LIN {X 0,Y 656.609,Z 179.375,A -85,B 0,C 180,E1 30688.866,E2 30688.866} C_VEL
LIN {X 0,Y 656.676,Z 179.373,A -85,B 0,C 180,E1 30685.897,E2 30685.897} C_VEL
LIN {X 0,Y 656.608,Z 179.376,A -85,B 0,C 180,E1 30683.091,E2 30683.091} C_VEL
LIN {X 0,Y 656.674,Z 179.374,A -85,B 0,C 180,E1 30680.271,E2 30680.271} C_VEL
LIN {X 0,Y 656.609,Z 179.374,A -85,B 0,C 180,E1 30677.335,E2 30677.335} C_VEL
LIN {X 0,Y 656.626,Z 179.376,A -85,B 0,C 180,E1 30674.728,E2 30674.728} C_VEL
LIN {X 0,Y 656.62,Z 179.375,A -85,B 0,C 180,E1 30671.568,E2 30671.568} C_VEL
LIN {X 0,Y 656.615,Z 179.375,A -85,B 0,C 180,E1 30668.941,E2 30668.941} C_VEL
LIN {X 0,Y 656.649,Z 179.375,A -85,B 0,C 180,E1 30665.919,E2 30665.919} C_VEL
LIN {X 0,Y 656.609,Z 179.373,A -85,B 0,C 180,E1 30663.173,E2 30663.173} C_VEL
LIN {X 0,Y 656.682,Z 179.373,A -85,B 0,C 180,E1 30660.216,E2 30660.216} C_VEL
LIN {X 0,Y 656.607,Z 179.374,A -85,B 0,C 180,E1 30657.365,E2 30657.365} C_VEL
LIN {X 0,Y 656.689,Z 179.372,A -85,B 0,C 180,E1 30654.398,E2 30654.398} C_VEL
LIN {X 0,Y 656.607,Z 179.374,A -85,B 0,C 180,E1 30651.483,E2 30651.483} C_VEL
LIN {X 0,Y 656.656,Z 179.373,A -85,B 0,C 180,E1 30648.758,E2 30648.758} C_VEL
LIN {X 0,Y 656.615,Z 179.374,A -85,B 0,C 180,E1 30645.786,E2 30645.786} C_VEL
LIN {X 0,Y 656.622,Z 179.374,A -85,B 0,C 180,E1 30643.136,E2 30643.136} C_VEL
LIN {X 0,Y 656.625,Z 179.373,A -85,B 0,C 180,E1 30639.987,E2 30639.987} C_VEL
LIN {X 0,Y 656.612,Z 179.372,A -85,B 0,C 180,E1 30637.364,E2 30637.364} C_VEL
LIN {X 0,Y 656.649,Z 179.359,A -85,B 0,C 180,E1 30634.292,E2 30634.292} C_VEL
LIN {X 0,Y 656.61,Z 179.373,A -85,B 0,C 180,E1 30631.591,E2 30631.591} C_VEL
LIN {X 0,Y 656.691,Z 179.343,A -85,B 0,C 180,E1 30628.661,E2 30628.661} C_VEL
LIN {X 0,Y 656.607,Z 179.365,A -85,B 0,C 180,E1 30625.722,E2 30625.722} C_VEL
LIN {X 0,Y 656.697,Z 179.367,A -85,B 0,C 180,E1 30622.752,E2 30622.752} C_VEL
LIN {X 0,Y 656.608,Z 179.372,A -85,B 0,C 180,E1 30619.852,E2 30619.852} C_VEL
LIN {X 0,Y 656.666,Z 179.366,A -85,B 0,C 180,E1 30617.038,E2 30617.038} C_VEL
LIN {X 0,Y 656.612,Z 179.371,A -85,B 0,C 180,E1 30614.095,E2 30614.095} C_VEL
LIN {X 0,Y 656.628,Z 179.365,A -85,B 0,C 180,E1 30611.418,E2 30611.418} C_VEL
LIN {X 0,Y 656.622,Z 179.367,A -85,B 0,C 180,E1 30608.318,E2 30608.318} C_VEL
LIN {X 0,Y 656.609,Z 179.37,A -85,B 0,C 180,E1 30605.768,E2 30605.768} C_VEL
LIN {X 0,Y 656.67,Z 179.363,A -85,B 0,C 180,E1 30602.793,E2 30602.793} C_VEL
LIN {X 0,Y 656.607,Z 179.372,A -85,B 0,C 180,E1 30600,E2 30600} C_VEL
LIN {X 0,Y 656.686,Z 179.363,A -85,B 0,C 180,E1 30597.086,E2 30597.086} C_VEL
LIN {X 0,Y 656.609,Z 179.371,A -85,B 0,C 180,E1 30594.144,E2 30594.144} C_VEL
LIN {X 0,Y 656.641,Z 179.362,A -85,B 0,C 180,E1 30591.506,E2 30591.506} C_VEL
LIN {X 0,Y 656.614,Z 179.368,A -85,B 0,C 180,E1 30588.404,E2 30588.404} C_VEL
LIN {X 0,Y 656.628,Z 179.369,A -85,B 0,C 180,E1 30585.718,E2 30585.718} C_VEL
LIN {X 0,Y 656.62,Z 179.365,A -85,B 0,C 180,E1 30582.543,E2 30582.543} C_VEL
LIN {X 0,Y 656.621,Z 179.372,A -85,B 0,C 180,E1 30579.87,E2 30579.87} C_VEL
LIN {X 0,Y 656.624,Z 179.372,A -85,B 0,C 180,E1 30576.651,E2 30576.651} C_VEL
LIN {X 0,Y 656.618,Z 179.369,A -85,B 0,C 180,E1 30573.988,E2 30573.988} C_VEL
LIN {X 0,Y 656.631,Z 179.359,A -85,B 0,C 180,E1 30570.838,E2 30570.838} C_VEL
LIN {X 0,Y 656.612,Z 179.372,A -85,B 0,C 180,E1 30568.204,E2 30568.204} C_VEL
LIN {X 0,Y 656.678,Z 179.356,A -85,B 0,C 180,E1 30565.286,E2 30565.286} C_VEL
LIN {X 0,Y 656.609,Z 179.373,A -85,B 0,C 180,E1 30562.474,E2 30562.474} C_VEL
LIN {X 0,Y 656.666,Z 179.36,A -85,B 0,C 180,E1 30559.674,E2 30559.674} C_VEL
LIN {X 0,Y 656.612,Z 179.369,A -85,B 0,C 180,E1 30556.702,E2 30556.702} C_VEL
LIN {X 0,Y 656.639,Z 179.373,A -85,B 0,C 180,E1 30553.969,E2 30553.969} C_VEL
LIN {X 0,Y 656.622,Z 179.376,A -85,B 0,C 180,E1 30550.897,E2 30550.897} C_VEL
LIN {X 0,Y 656.614,Z 179.346,A -85,B 0,C 180,E1 30548.294,E2 30548.294} C_VEL
LIN {X 0,Y 656.638,Z 179.375,A -85,B 0,C 180,E1 30545.143,E2 30545.143} C_VEL
LIN {X 0,Y 656.711,Z 179.583,A -85,B 0,C 180,E1 30543.756,E2 30543.756} C_VEL
LIN {X 0,Y 663.323,Z 201.913,A -85,B 0,C 180,E1 30541.387,E2 30541.387} C_VEL
LIN {X 0,Y 662.57,Z 225.531,A -85,B 0,C 180,E1 30539.388,E2 30539.388} C_VEL
LIN {X 0,Y 667.017,Z 246.185,A -85,B 0,C 180,E1 30538.921,E2 30538.921} C_VEL
LIN {X 0,Y 664.801,Z 516.791,A -85,B 0,C 180,E1 30535.804,E2 30535.804} C_VEL
LIN {X 0,Y 664.373,Z 539.375,A -85,B 0,C 180,E1 30535.464,E2 30535.464} C_VEL
LIN {X 0,Y 663.94,Z 557.307,A -85,B 0,C 180,E1 30535.08,E2 30535.08} C_VEL
LIN {X 0,Y 663.439,Z 573.967,A -85,B 0,C 180,E1 30534.624,E2 30534.624} C_VEL
LIN {X 0,Y 662.861,Z 590.358,A -85,B 0,C 180,E1 30534.078,E2 30534.078} C_VEL
LIN {X 0,Y 662.199,Z 606.836,A -85,B 0,C 180,E1 30533.424,E2 30533.424} C_VEL
LIN {X 0,Y 661.522,Z 623.1,A -85,B 0,C 180,E1 30532.667,E2 30532.667} C_VEL
LIN {X 0,Y 660.779,Z 639.904,A -85,B 0,C 180,E1 30531.758,E2 30531.758} C_VEL
LIN {X 0,Y 659.792,Z 660.39,A -85,B 0,C 180,E1 30530.442,E2 30530.442} C_VEL
LIN {X 0,Y 659.062,Z 675.422,A -85,B 0,C 180,E1 30529.311,E2 30529.311} C_VEL
LIN {X 0,Y 658.429,Z 688.648,A -85,B 0,C 180,E1 30528.182,E2 30528.182} C_VEL
LIN {X 0,Y 657.872,Z 701.254,A -85,B 0,C 180,E1 30526.964,E2 30526.964} C_VEL
LIN {X 0,Y 657.324,Z 714.341,A -85,B 0,C 180,E1 30525.527,E2 30525.527} C_VEL
LIN {X 0,Y 656.796,Z 728.196,A -85,B 0,C 180,E1 30523.737,E2 30523.737} C_VEL
LIN {X 0,Y 656.462,Z 738.682,A -85,B 0,C 180,E1 30522.132,E2 30522.132} C_VEL
LIN {X 0,Y 656.245,Z 747.113,A -85,B 0,C 180,E1 30520.622,E2 30520.622} C_VEL
LIN {X 0,Y 656.073,Z 755.438,A -85,B 0,C 180,E1 30518.853,E2 30518.853} C_VEL
LIN {X 0,Y 655.962,Z 762.536,A -85,B 0,C 180,E1 30516.915,E2 30516.915} C_VEL
LIN {X 0,Y 655.927,Z 767.164,A -85,B 0,C 180,E1 30515.247,E2 30515.247} C_VEL
LIN {X 0,Y 655.919,Z 770.374,A -85,B 0,C 180,E1 30513.67,E2 30513.67} C_VEL
LIN {X 0,Y 655.916,Z 772.695,A -85,B 0,C 180,E1 30511.834,E2 30511.834} C_VEL
LIN {X 0,Y 655.903,Z 773.44,A -85,B 0,C 180,E1 30509.738,E2 30509.738} C_VEL
LIN {X 0,Y 655.913,Z 772.434,A -85,B 0,C 180,E1 30507.904,E2 30507.904} C_VEL
LIN {X 0,Y 655.922,Z 770.083,A -85,B 0,C 180,E1 30506.155,E2 30506.155} C_VEL
LIN {X 0,Y 655.941,Z 766.135,A -85,B 0,C 180,E1 30504.314,E2 30504.314} C_VEL
LIN {X 0,Y 655.999,Z 759.842,A -85,B 0,C 180,E1 30502.293,E2 30502.293} C_VEL
LIN {X 0,Y 656.109,Z 753.065,A -85,B 0,C 180,E1 30500.616,E2 30500.616} C_VEL
LIN {X 0,Y 656.274,Z 745.72,A -85,B 0,C 180,E1 30499.111,E2 30499.111} C_VEL
LIN {X 0,Y 656.555,Z 735.998,A -85,B 0,C 180,E1 30497.423,E2 30497.423} C_VEL
LIN {X 0,Y 656.97,Z 723.616,A -85,B 0,C 180,E1 30495.638,E2 30495.638} C_VEL
LIN {X 0,Y 657.408,Z 711.981,A -85,B 0,C 180,E1 30494.204,E2 30494.204} C_VEL
LIN {X 0,Y 657.918,Z 700.216,A -85,B 0,C 180,E1 30492.93,E2 30492.93} C_VEL
LIN {X 0,Y 658.499,Z 687.157,A -85,B 0,C 180,E1 30491.683,E2 30491.683} C_VEL
LIN {X 0,Y 659.331,Z 670.387,A -85,B 0,C 180,E1 30490.283,E2 30490.283} C_VEL
LIN {X 0,Y 660.165,Z 652.635,A -85,B 0,C 180,E1 30489.033,E2 30489.033} C_VEL
LIN {X 0,Y 660.876,Z 637.494,A -85,B 0,C 180,E1 30488.106,E2 30488.106} C_VEL
LIN {X 0,Y 661.557,Z 622.179,A -85,B 0,C 180,E1 30487.287,E2 30487.287} C_VEL
LIN {X 0,Y 662.229,Z 606.166,A -85,B 0,C 180,E1 30486.547,E2 30486.547} C_VEL
LIN {X 0,Y 662.861,Z 590.357,A -85,B 0,C 180,E1 30485.922,E2 30485.922} C_VEL
LIN {X 0,Y 663.439,Z 573.966,A -85,B 0,C 180,E1 30485.376,E2 30485.376} C_VEL
LIN {X 0,Y 663.961,Z 556.505,A -85,B 0,C 180,E1 30484.9,E2 30484.9} C_VEL
LIN {X 0,Y 664.453,Z 536.479,A -85,B 0,C 180,E1 30484.481,E2 30484.481} C_VEL
LIN {X 0,Y 664.876,Z 507.354,A -85,B 0,C 180,E1 30484.089,E2 30484.089} C_VEL
LIN {X 0,Y 667.019,Z 245.178,A -85,B 0,C 180,E1 30481.067,E2 30481.067} C_VEL
LIN {X 0,Y 662.536,Z 225.127,A -85,B 0,C 180,E1 30480.591,E2 30480.591} C_VEL
LIN {X 0,Y 663.211,Z 201.553,A -85,B 0,C 180,E1 30478.576,E2 30478.576} C_VEL
LIN {X 0,Y 656.698,Z 179.514,A -85,B 0,C 180,E1 30476.226,E2 30476.226} C_VEL
LIN {X 0,Y 656.607,Z 179.349,A -85,B 0,C 180,E1 30473.355,E2 30473.355} C_VEL
LIN {X 0,Y 656.694,Z 179.36,A -85,B 0,C 180,E1 30470.394,E2 30470.394} C_VEL
LIN {X 0,Y 656.609,Z 179.368,A -85,B 0,C 180,E1 30467.48,E2 30467.48} C_VEL
LIN {X 0,Y 656.686,Z 179.361,A -85,B 0,C 180,E1 30464.562,E2 30464.562} C_VEL
LIN {X 0,Y 656.611,Z 179.372,A -85,B 0,C 180,E1 30461.602,E2 30461.602} C_VEL
LIN {X 0,Y 656.657,Z 179.364,A -85,B 0,C 180,E1 30458.855,E2 30458.855} C_VEL
LIN {X 0,Y 656.617,Z 179.364,A -85,B 0,C 180,E1 30455.893,E2 30455.893} C_VEL
LIN {X 0,Y 656.622,Z 179.368,A -85,B 0,C 180,E1 30453.244,E2 30453.244} C_VEL
LIN {X 0,Y 656.625,Z 179.361,A -85,B 0,C 180,E1 30450.066,E2 30450.066} C_VEL
LIN {X 0,Y 656.614,Z 179.351,A -85,B 0,C 180,E1 30447.418,E2 30447.418} C_VEL
LIN {X 0,Y 656.65,Z 179.372,A -85,B 0,C 180,E1 30444.372,E2 30444.372} C_VEL
LIN {X 0,Y 656.607,Z 179.366,A -85,B 0,C 180,E1 30441.718,E2 30441.718} C_VEL
LIN {X 0,Y 656.689,Z 179.368,A -85,B 0,C 180,E1 30438.832,E2 30438.832} C_VEL
LIN {X 0,Y 656.609,Z 179.371,A -85,B 0,C 180,E1 30435.909,E2 30435.909} C_VEL
LIN {X 0,Y 656.636,Z 179.368,A -85,B 0,C 180,E1 30433.293,E2 30433.293} C_VEL
LIN {X 0,Y 656.616,Z 179.371,A -85,B 0,C 180,E1 30430.174,E2 30430.174} C_VEL
LIN {X 0,Y 656.621,Z 179.363,A -85,B 0,C 180,E1 30427.525,E2 30427.525} C_VEL
LIN {X 0,Y 656.625,Z 179.369,A -85,B 0,C 180,E1 30424.367,E2 30424.367} C_VEL
LIN {X 0,Y 656.612,Z 179.368,A -85,B 0,C 180,E1 30421.745,E2 30421.745} C_VEL
LIN {X 0,Y 656.664,Z 179.364,A -85,B 0,C 180,E1 30418.779,E2 30418.779} C_VEL
LIN {X 0,Y 656.606,Z 179.372,A -85,B 0,C 180,E1 30415.983,E2 30415.983} C_VEL
LIN {X 0,Y 656.691,Z 179.363,A -85,B 0,C 180,E1 30413.003,E2 30413.003} C_VEL
LIN {X 0,Y 656.608,Z 179.372,A -85,B 0,C 180,E1 30410.091,E2 30410.091} C_VEL
LIN {X 0,Y 656.69,Z 179.364,A -85,B 0,C 180,E1 30407.156,E2 30407.156} C_VEL
LIN {X 0,Y 656.608,Z 179.37,A -85,B 0,C 180,E1 30404.273,E2 30404.273} C_VEL
LIN {X 0,Y 656.65,Z 179.369,A -85,B 0,C 180,E1 30401.535,E2 30401.535} C_VEL
LIN {X 0,Y 656.614,Z 179.366,A -85,B 0,C 180,E1 30398.482,E2 30398.482} C_VEL
LIN {X 0,Y 656.619,Z 179.373,A -85,B 0,C 180,E1 30395.914,E2 30395.914} C_VEL
LIN {X 0,Y 656.622,Z 179.344,A -85,B 0,C 180,E1 30392.719,E2 30392.719} C_VEL
LIN {X 0,Y 656.61,Z 179.366,A -85,B 0,C 180,E1 30390.135,E2 30390.135} C_VEL
LIN {X 0,Y 656.67,Z 179.365,A -85,B 0,C 180,E1 30387.175,E2 30387.175} C_VEL
LIN {X 0,Y 656.603,Z 179.355,A -85,B 0,C 180,E1 30384.321,E2 30384.321} C_VEL
LIN {X 0,Y 656.691,Z 179.372,A -85,B 0,C 180,E1 30381.352,E2 30381.352} C_VEL
LIN {X 0,Y 656.608,Z 179.373,A -85,B 0,C 180,E1 30380.38,E2 30380.38} C_VEL
LIN {X 0,Y 655.64,Z 179.501,A -85,B 0,C 180,E1 30379.708,E2 30379.708} C_VEL
LIN {X 0,Y 649.202,Z 180.307,A -85,B 0,C 180,E1 30377.775,E2 30377.775} C_VEL
LIN {X 0,Y 648.739,Z 180.362,A -85,B 0,C 180,E1 30377.334,E2 30377.334} C_VEL
LIN {X 0,Y 648.669,Z 180.363,A -85,B 0,C 180,E1 30374.464,E2 30374.464} C_VEL
LIN {X 0,Y 648.756,Z 180.361,A -85,B 0,C 180,E1 30371.492,E2 30371.492} C_VEL
LIN {X 0,Y 648.668,Z 180.363,A -85,B 0,C 180,E1 30368.6,E2 30368.6} C_VEL
LIN {X 0,Y 648.743,Z 180.362,A -85,B 0,C 180,E1 30365.683,E2 30365.683} C_VEL
LIN {X 0,Y 648.669,Z 180.363,A -85,B 0,C 180,E1 30362.687,E2 30362.687} C_VEL
LIN {X 0,Y 648.741,Z 180.362,A -85,B 0,C 180,E1 30359.803,E2 30359.803} C_VEL
LIN {X 0,Y 648.67,Z 180.362,A -85,B 0,C 180,E1 30356.811,E2 30356.811} C_VEL
LIN {X 0,Y 648.721,Z 180.363,A -85,B 0,C 180,E1 30354.007,E2 30354.007} C_VEL
LIN {X 0,Y 648.676,Z 180.364,A -85,B 0,C 180,E1 30351.045,E2 30351.045} C_VEL
LIN {X 0,Y 648.691,Z 180.364,A -85,B 0,C 180,E1 30348.325,E2 30348.325} C_VEL
LIN {X 0,Y 648.68,Z 180.365,A -85,B 0,C 180,E1 30345.189,E2 30345.189} C_VEL
LIN {X 0,Y 648.677,Z 180.363,A -85,B 0,C 180,E1 30342.551,E2 30342.551} C_VEL
LIN {X 0,Y 648.692,Z 180.363,A -85,B 0,C 180,E1 30339.402,E2 30339.402} C_VEL
LIN {X 0,Y 648.671,Z 180.365,A -85,B 0,C 180,E1 30336.727,E2 30336.727} C_VEL
LIN {X 0,Y 648.72,Z 180.362,A -85,B 0,C 180,E1 30333.711,E2 30333.711} C_VEL
LIN {X 0,Y 648.669,Z 180.365,A -85,B 0,C 180,E1 30330.883,E2 30330.883} C_VEL
LIN {X 0,Y 648.747,Z 180.359,A -85,B 0,C 180,E1 30327.969,E2 30327.969} C_VEL
LIN {X 0,Y 648.668,Z 180.364,A -85,B 0,C 180,E1 30325.049,E2 30325.049} C_VEL
LIN {X 0,Y 648.756,Z 180.359,A -85,B 0,C 180,E1 30322.117,E2 30322.117} C_VEL
LIN {X 0,Y 648.669,Z 180.365,A -85,B 0,C 180,E1 30319.162,E2 30319.162} C_VEL
LIN {X 0,Y 648.755,Z 180.36,A -85,B 0,C 180,E1 30316.181,E2 30316.181} C_VEL
LIN {X 0,Y 648.669,Z 180.363,A -85,B 0,C 180,E1 30313.249,E2 30313.249} C_VEL
LIN {X 0,Y 648.742,Z 180.36,A -85,B 0,C 180,E1 30310.343,E2 30310.343} C_VEL
LIN {X 0,Y 648.672,Z 180.364,A -85,B 0,C 180,E1 30307.418,E2 30307.418} C_VEL
LIN {X 0,Y 648.699,Z 180.364,A -85,B 0,C 180,E1 30304.729,E2 30304.729} C_VEL
LIN {X 0,Y 648.679,Z 180.364,A -85,B 0,C 180,E1 30301.661,E2 30301.661} C_VEL
LIN {X 0,Y 648.673,Z 180.363,A -85,B 0,C 180,E1 30299.121,E2 30299.121} C_VEL
LIN {X 0,Y 648.718,Z 180.363,A -85,B 0,C 180,E1 30296.09,E2 30296.09} C_VEL
LIN {X 0,Y 648.672,Z 180.362,A -85,B 0,C 180,E1 30293.273,E2 30293.273} C_VEL
LIN {X 0,Y 648.735,Z 180.362,A -85,B 0,C 180,E1 30290.274,E2 30290.274} C_VEL
LIN {X 0,Y 648.669,Z 180.363,A -85,B 0,C 180,E1 30287.461,E2 30287.461} C_VEL
LIN {X 0,Y 648.748,Z 180.361,A -85,B 0,C 180,E1 30284.479,E2 30284.479} C_VEL
LIN {X 0,Y 648.671,Z 180.362,A -85,B 0,C 180,E1 30281.626,E2 30281.626} C_VEL
LIN {X 0,Y 648.713,Z 180.362,A -85,B 0,C 180,E1 30278.897,E2 30278.897} C_VEL
LIN {X 0,Y 648.671,Z 180.343,A -85,B 0,C 180,E1 30275.837,E2 30275.837} C_VEL
LIN {X 0,Y 648.688,Z 180.354,A -85,B 0,C 180,E1 30273.175,E2 30273.175} C_VEL
LIN {X 0,Y 648.683,Z 180.354,A -85,B 0,C 180,E1 30270.064,E2 30270.064} C_VEL
LIN {X 0,Y 648.674,Z 180.329,A -85,B 0,C 180,E1 30267.409,E2 30267.409} C_VEL
LIN {X 0,Y 648.701,Z 180.362,A -85,B 0,C 180,E1 30264.302,E2 30264.302} C_VEL
LIN {X 0,Y 648.669,Z 180.355,A -85,B 0,C 180,E1 30261.617,E2 30261.617} C_VEL
LIN {X 0,Y 648.744,Z 180.358,A -85,B 0,C 180,E1 30258.698,E2 30258.698} C_VEL
LIN {X 0,Y 648.667,Z 180.358,A -85,B 0,C 180,E1 30255.833,E2 30255.833} C_VEL
LIN {X 0,Y 648.738,Z 180.356,A -85,B 0,C 180,E1 30253.005,E2 30253.005} C_VEL
LIN {X 0,Y 648.671,Z 180.361,A -85,B 0,C 180,E1 30249.987,E2 30249.987} C_VEL
LIN {X 0,Y 648.723,Z 180.353,A -85,B 0,C 180,E1 30247.172,E2 30247.172} C_VEL
LIN {X 0,Y 648.671,Z 180.361,A -85,B 0,C 180,E1 30244.155,E2 30244.155} C_VEL
LIN {X 0,Y 648.7,Z 180.352,A -85,B 0,C 180,E1 30241.413,E2 30241.413} C_VEL
LIN {X 0,Y 648.677,Z 180.357,A -85,B 0,C 180,E1 30238.322,E2 30238.322} C_VEL
LIN {X 0,Y 648.69,Z 180.357,A -85,B 0,C 180,E1 30235.58,E2 30235.58} C_VEL
LIN {X 0,Y 648.682,Z 180.35,A -85,B 0,C 180,E1 30232.471,E2 30232.471} C_VEL
LIN {X 0,Y 648.679,Z 180.36,A -85,B 0,C 180,E1 30229.789,E2 30229.789} C_VEL
LIN {X 0,Y 648.691,Z 180.358,A -85,B 0,C 180,E1 30226.632,E2 30226.632} C_VEL
LIN {X 0,Y 648.672,Z 180.361,A -85,B 0,C 180,E1 30224.075,E2 30224.075} C_VEL
LIN {X 0,Y 648.743,Z 180.359,A -85,B 0,C 180,E1 30221.115,E2 30221.115} C_VEL
LIN {X 0,Y 648.67,Z 180.355,A -85,B 0,C 180,E1 30218.287,E2 30218.287} C_VEL
LIN {X 0,Y 648.742,Z 180.361,A -85,B 0,C 180,E1 30215.408,E2 30215.408} C_VEL
LIN {X 0,Y 648.669,Z 180.339,A -85,B 0,C 180,E1 30212.455,E2 30212.455} C_VEL
LIN {X 0,Y 648.705,Z 180.349,A -85,B 0,C 180,E1 30209.733,E2 30209.733} C_VEL
LIN {X 0,Y 648.678,Z 180.356,A -85,B 0,C 180,E1 30206.651,E2 30206.651} C_VEL
LIN {X 0,Y 648.691,Z 180.352,A -85,B 0,C 180,E1 30203.927,E2 30203.927} C_VEL
LIN {X 0,Y 648.681,Z 180.352,A -85,B 0,C 180,E1 30200.803,E2 30200.803} C_VEL
LIN {X 0,Y 648.676,Z 180.361,A -85,B 0,C 180,E1 30198.241,E2 30198.241} C_VEL
LIN {X 0,Y 648.71,Z 180.356,A -85,B 0,C 180,E1 30195.147,E2 30195.147} C_VEL
LIN {X 0,Y 648.672,Z 180.357,A -85,B 0,C 180,E1 30192.409,E2 30192.409} C_VEL
LIN {X 0,Y 648.742,Z 180.346,A -85,B 0,C 180,E1 30189.45,E2 30189.45} C_VEL
LIN {X 0,Y 648.668,Z 180.336,A -85,B 0,C 180,E1 30186.573,E2 30186.573} C_VEL
LIN {X 0,Y 648.721,Z 180.544,A -85,B 0,C 180,E1 30184.123,E2 30184.123} C_VEL
LIN {X 0,Y 655.582,Z 203.464,A -85,B 0,C 180,E1 30181.641,E2 30181.641} C_VEL
LIN {X 0,Y 655.853,Z 206.269,A -85,B 0,C 180,E1 30181.377,E2 30181.377} C_VEL
LIN {X 0,Y 655.176,Z 225.339,A -85,B 0,C 180,E1 30179.753,E2 30179.753} C_VEL
LIN {X 0,Y 659.991,Z 247.608,A -85,B 0,C 180,E1 30179.239,E2 30179.239} C_VEL
LIN {X 0,Y 657.572,Z 517.906,A -85,B 0,C 180,E1 30176.092,E2 30176.092} C_VEL
LIN {X 0,Y 657.117,Z 539.692,A -85,B 0,C 180,E1 30175.756,E2 30175.756} C_VEL
LIN {X 0,Y 656.647,Z 557.475,A -85,B 0,C 180,E1 30175.369,E2 30175.369} C_VEL
LIN {X 0,Y 656.088,Z 574.535,A -85,B 0,C 180,E1 30174.895,E2 30174.895} C_VEL
LIN {X 0,Y 655.488,Z 590.18,A -85,B 0,C 180,E1 30174.366,E2 30174.366} C_VEL
LIN {X 0,Y 654.779,Z 606.59,A -85,B 0,C 180,E1 30173.709,E2 30173.709} C_VEL
LIN {X 0,Y 654.071,Z 622.002,A -85,B 0,C 180,E1 30172.988,E2 30172.988} C_VEL
LIN {X 0,Y 653.293,Z 638.152,A -85,B 0,C 180,E1 30172.115,E2 30172.115} C_VEL
LIN {X 0,Y 652.35,Z 657.185,A -85,B 0,C 180,E1 30170.921,E2 30170.921} C_VEL
LIN {X 0,Y 651.442,Z 674.299,A -85,B 0,C 180,E1 30169.639,E2 30169.639} C_VEL
LIN {X 0,Y 650.738,Z 687.646,A -85,B 0,C 180,E1 30168.497,E2 30168.497} C_VEL
LIN {X 0,Y 650.113,Z 700.36,A -85,B 0,C 180,E1 30167.265,E2 30167.265} C_VEL
LIN {X 0,Y 649.567,Z 711.975,A -85,B 0,C 180,E1 30165.992,E2 30165.992} C_VEL
LIN {X 0,Y 649.058,Z 724.307,A -85,B 0,C 180,E1 30164.45,E2 30164.45} C_VEL
LIN {X 0,Y 648.597,Z 736.683,A -85,B 0,C 180,E1 30162.617,E2 30162.617} C_VEL
LIN {X 0,Y 648.311,Z 745.717,A -85,B 0,C 180,E1 30161.024,E2 30161.024} C_VEL
LIN {X 0,Y 648.131,Z 753.06,A -85,B 0,C 180,E1 30159.5,E2 30159.5} C_VEL
LIN {X 0,Y 648.01,Z 759.836,A -85,B 0,C 180,E1 30157.803,E2 30157.803} C_VEL
LIN {X 0,Y 647.947,Z 765.927,A -85,B 0,C 180,E1 30155.845,E2 30155.845} C_VEL
LIN {X 0,Y 647.923,Z 769.932,A -85,B 0,C 180,E1 30153.982,E2 30153.982} C_VEL
LIN {X 0,Y 647.909,Z 772.254,A -85,B 0,C 180,E1 30152.299,E2 30152.299} C_VEL
LIN {X 0,Y 647.903,Z 773.327,A -85,B 0,C 180,E1 30150.619,E2 30150.619} C_VEL
LIN {X 0,Y 647.902,Z 773.153,A -85,B 0,C 180,E1 30148.851,E2 30148.851} C_VEL
LIN {X 0,Y 647.904,Z 771.099,A -85,B 0,C 180,E1 30146.727,E2 30146.727} C_VEL
LIN {X 0,Y 647.917,Z 767.778,A -85,B 0,C 180,E1 30144.954,E2 30144.954} C_VEL
LIN {X 0,Y 647.958,Z 763.598,A -85,B 0,C 180,E1 30143.355,E2 30143.355} C_VEL
LIN {X 0,Y 648.049,Z 757.856,A -85,B 0,C 180,E1 30141.662,E2 30141.662} C_VEL
LIN {X 0,Y 648.235,Z 749.423,A -85,B 0,C 180,E1 30139.694,E2 30139.694} C_VEL
LIN {X 0,Y 648.489,Z 739.748,A -85,B 0,C 180,E1 30137.897,E2 30137.897} C_VEL
LIN {X 0,Y 648.822,Z 730.029,A -85,B 0,C 180,E1 30136.364,E2 30136.364} C_VEL
LIN {X 0,Y 649.247,Z 719.431,A -85,B 0,C 180,E1 30134.916,E2 30134.916} C_VEL
LIN {X 0,Y 649.876,Z 705.645,A -85,B 0,C 180,E1 30133.281,E2 30133.281} C_VEL
LIN {X 0,Y 650.594,Z 690.538,A -85,B 0,C 180,E1 30131.769,E2 30131.769} C_VEL
LIN {X 0,Y 651.287,Z 677.089,A -85,B 0,C 180,E1 30130.589,E2 30130.589} C_VEL
LIN {X 0,Y 651.98,Z 663.838,A -85,B 0,C 180,E1 30129.561,E2 30129.561} C_VEL
LIN {X 0,Y 652.719,Z 649.399,A -85,B 0,C 180,E1 30128.574,E2 30128.574} C_VEL
LIN {X 0,Y 653.476,Z 634.276,A -85,B 0,C 180,E1 30127.664,E2 30127.664} C_VEL
LIN {X 0,Y 654.308,Z 617.395,A -85,B 0,C 180,E1 30126.783,E2 30126.783} C_VEL
LIN {X 0,Y 655.285,Z 595.284,A -85,B 0,C 180,E1 30125.822,E2 30125.822} C_VEL
LIN {X 0,Y 656.006,Z 576.766,A -85,B 0,C 180,E1 30125.174,E2 30125.174} C_VEL
LIN {X 0,Y 656.593,Z 559.359,A -85,B 0,C 180,E1 30124.679,E2 30124.679} C_VEL
LIN {X 0,Y 657.058,Z 542.385,A -85,B 0,C 180,E1 30124.297,E2 30124.297} C_VEL
LIN {X 0,Y 657.429,Z 525.016,A -85,B 0,C 180,E1 30124.007,E2 30124.007} C_VEL
LIN {X 0,Y 659.812,Z 267.465,A -85,B 0,C 180,E1 30120.995,E2 30120.995} C_VEL
LIN {X 0,Y 659.802,Z 245.831,A -85,B 0,C 180,E1 30120.73,E2 30120.73} C_VEL
LIN {X 0,Y 655.119,Z 224.707,A -85,B 0,C 180,E1 30120.216,E2 30120.216} C_VEL
LIN {X 0,Y 655.742,Z 204.05,A -85,B 0,C 180,E1 30118.419,E2 30118.419} C_VEL
LIN {X 0,Y 649.083,Z 181.929,A -85,B 0,C 180,E1 30116.052,E2 30116.052} C_VEL
LIN {X 0,Y 648.713,Z 180.503,A -85,B 0,C 180,E1 30115.864,E2 30115.864} C_VEL
LIN {X 0,Y 648.674,Z 180.329,A -85,B 0,C 180,E1 30113.131,E2 30113.131} C_VEL
LIN {X 0,Y 648.702,Z 180.366,A -85,B 0,C 180,E1 30110.002,E2 30110.002} C_VEL
LIN {X 0,Y 648.673,Z 180.357,A -85,B 0,C 180,E1 30107.302,E2 30107.302} C_VEL
LIN {X 0,Y 648.73,Z 180.35,A -85,B 0,C 180,E1 30104.284,E2 30104.284} C_VEL
LIN {X 0,Y 648.671,Z 180.361,A -85,B 0,C 180,E1 30101.493,E2 30101.493} C_VEL
LIN {X 0,Y 648.756,Z 180.352,A -85,B 0,C 180,E1 30098.62,E2 30098.62} C_VEL
LIN {X 0,Y 648.669,Z 180.352,A -85,B 0,C 180,E1 30095.639,E2 30095.639} C_VEL
LIN {X 0,Y 648.748,Z 180.357,A -85,B 0,C 180,E1 30092.71,E2 30092.71} C_VEL
LIN {X 0,Y 648.67,Z 180.349,A -85,B 0,C 180,E1 30089.759,E2 30089.759} C_VEL
LIN {X 0,Y 648.722,Z 180.339,A -85,B 0,C 180,E1 30086.946,E2 30086.946} C_VEL
LIN {X 0,Y 648.674,Z 180.361,A -85,B 0,C 180,E1 30083.916,E2 30083.916} C_VEL
LIN {X 0,Y 648.695,Z 180.354,A -85,B 0,C 180,E1 30081.237,E2 30081.237} C_VEL
LIN {X 0,Y 648.683,Z 180.353,A -85,B 0,C 180,E1 30078.142,E2 30078.142} C_VEL
LIN {X 0,Y 648.682,Z 180.359,A -85,B 0,C 180,E1 30075.466,E2 30075.466} C_VEL
LIN {X 0,Y 648.686,Z 180.357,A -85,B 0,C 180,E1 30072.28,E2 30072.28} C_VEL
LIN {X 0,Y 648.678,Z 180.36,A -85,B 0,C 180,E1 30069.583,E2 30069.583} C_VEL
LIN {X 0,Y 648.697,Z 180.361,A -85,B 0,C 180,E1 30066.461,E2 30066.461} C_VEL
LIN {X 0,Y 648.67,Z 180.358,A -85,B 0,C 180,E1 30063.801,E2 30063.801} C_VEL
LIN {X 0,Y 648.731,Z 180.361,A -85,B 0,C 180,E1 30060.795,E2 30060.795} C_VEL
LIN {X 0,Y 648.668,Z 180.353,A -85,B 0,C 180,E1 30057.968,E2 30057.968} C_VEL
LIN {X 0,Y 648.749,Z 180.361,A -85,B 0,C 180,E1 30055.049,E2 30055.049} C_VEL
LIN {X 0,Y 648.67,Z 180.356,A -85,B 0,C 180,E1 30052.204,E2 30052.204} C_VEL
LIN {X 0,Y 648.715,Z 180.361,A -85,B 0,C 180,E1 30049.431,E2 30049.431} C_VEL
LIN {X 0,Y 648.673,Z 180.361,A -85,B 0,C 180,E1 30046.359,E2 30046.359} C_VEL
LIN {X 0,Y 648.683,Z 180.359,A -85,B 0,C 180,E1 30043.775,E2 30043.775} C_VEL
LIN {X 0,Y 648.68,Z 180.361,A -85,B 0,C 180,E1 30040.552,E2 30040.552} C_VEL
LIN {X 0,Y 648.683,Z 180.355,A -85,B 0,C 180,E1 30037.86,E2 30037.86} C_VEL
LIN {X 0,Y 648.681,Z 180.354,A -85,B 0,C 180,E1 30034.627,E2 30034.627} C_VEL
LIN {X 0,Y 648.679,Z 180.331,A -85,B 0,C 180,E1 30031.957,E2 30031.957} C_VEL
LIN {X 0,Y 648.689,Z 180.362,A -85,B 0,C 180,E1 30028.8,E2 30028.8} C_VEL
LIN {X 0,Y 648.673,Z 180.353,A -85,B 0,C 180,E1 30026.173,E2 30026.173} C_VEL
LIN {X 0,Y 648.716,Z 180.356,A -85,B 0,C 180,E1 30023.115,E2 30023.115} C_VEL
LIN {X 0,Y 648.67,Z 180.362,A -85,B 0,C 180,E1 30020.345,E2 30020.345} C_VEL
LIN {X 0,Y 648.748,Z 180.361,A -85,B 0,C 180,E1 30017.42,E2 30017.42} C_VEL
LIN {X 0,Y 648.739,Z 180.362,A -85,B 0,C 180,E1 30017.334,E2 30017.334} C_VEL
LIN {X 0,Y 647.695,Z 180.49,A -85,B 0,C 180,E1 30016.653,E2 30016.653} C_VEL
LIN {X 0,Y 641.24,Z 181.29,A -85,B 0,C 180,E1 30014.746,E2 30014.746} C_VEL
LIN {X 0,Y 640.736,Z 181.352,A -85,B 0,C 180,E1 30014.25,E2 30014.25} C_VEL
LIN {X 0,Y 640.769,Z 181.351,A -85,B 0,C 180,E1 30011.179,E2 30011.179} C_VEL
LIN {X 0,Y 640.732,Z 181.352,A -85,B 0,C 180,E1 30008.427,E2 30008.427} C_VEL
LIN {X 0,Y 640.798,Z 181.35,A -85,B 0,C 180,E1 30005.46,E2 30005.46} C_VEL
LIN {X 0,Y 640.731,Z 181.353,A -85,B 0,C 180,E1 30002.569,E2 30002.569} C_VEL
LIN {X 0,Y 640.818,Z 181.347,A -85,B 0,C 180,E1 29999.641,E2 29999.641} C_VEL
LIN {X 0,Y 640.731,Z 181.352,A -85,B 0,C 180,E1 29996.704,E2 29996.704} C_VEL
LIN {X 0,Y 640.813,Z 181.348,A -85,B 0,C 180,E1 29993.735,E2 29993.735} C_VEL
LIN {X 0,Y 640.73,Z 181.353,A -85,B 0,C 180,E1 29990.809,E2 29990.809} C_VEL
LIN {X 0,Y 640.808,Z 181.349,A -85,B 0,C 180,E1 29987.857,E2 29987.857} C_VEL
LIN {X 0,Y 640.73,Z 181.354,A -85,B 0,C 180,E1 29984.919,E2 29984.919} C_VEL
LIN {X 0,Y 640.789,Z 181.352,A -85,B 0,C 180,E1 29982.068,E2 29982.068} C_VEL
LIN {X 0,Y 640.732,Z 181.353,A -85,B 0,C 180,E1 29979.067,E2 29979.067} C_VEL
LIN {X 0,Y 640.76,Z 181.354,A -85,B 0,C 180,E1 29976.36,E2 29976.36} C_VEL
LIN {X 0,Y 640.736,Z 181.354,A -85,B 0,C 180,E1 29973.22,E2 29973.22} C_VEL
LIN {X 0,Y 640.757,Z 181.352,A -85,B 0,C 180,E1 29970.447,E2 29970.447} C_VEL
LIN {X 0,Y 640.737,Z 181.354,A -85,B 0,C 180,E1 29967.317,E2 29967.317} C_VEL
LIN {X 0,Y 640.757,Z 181.353,A -85,B 0,C 180,E1 29964.539,E2 29964.539} C_VEL
LIN {X 0,Y 640.737,Z 181.353,A -85,B 0,C 180,E1 29961.385,E2 29961.385} C_VEL
LIN {X 0,Y 640.751,Z 181.354,A -85,B 0,C 180,E1 29958.662,E2 29958.662} C_VEL
LIN {X 0,Y 640.744,Z 181.354,A -85,B 0,C 180,E1 29955.543,E2 29955.543} C_VEL
LIN {X 0,Y 640.741,Z 181.353,A -85,B 0,C 180,E1 29952.849,E2 29952.849} C_VEL
LIN {X 0,Y 640.746,Z 181.353,A -85,B 0,C 180,E1 29949.638,E2 29949.638} C_VEL
LIN {X 0,Y 640.737,Z 181.353,A -85,B 0,C 180,E1 29947.031,E2 29947.031} C_VEL
LIN {X 0,Y 640.778,Z 181.351,A -85,B 0,C 180,E1 29943.997,E2 29943.997} C_VEL
LIN {X 0,Y 640.733,Z 181.353,A -85,B 0,C 180,E1 29941.175,E2 29941.175} C_VEL
LIN {X 0,Y 640.793,Z 181.35,A -85,B 0,C 180,E1 29938.174,E2 29938.174} C_VEL
LIN {X 0,Y 640.73,Z 181.353,A -85,B 0,C 180,E1 29935.327,E2 29935.327} C_VEL
LIN {X 0,Y 640.801,Z 181.35,A -85,B 0,C 180,E1 29932.296,E2 29932.296} C_VEL
LIN {X 0,Y 640.731,Z 181.351,A -85,B 0,C 180,E1 29929.463,E2 29929.463} C_VEL
LIN {X 0,Y 640.809,Z 181.349,A -85,B 0,C 180,E1 29926.516,E2 29926.516} C_VEL
LIN {X 0,Y 640.732,Z 181.352,A -85,B 0,C 180,E1 29923.611,E2 29923.611} C_VEL
LIN {X 0,Y 640.801,Z 181.351,A -85,B 0,C 180,E1 29920.691,E2 29920.691} C_VEL
LIN {X 0,Y 640.732,Z 181.35,A -85,B 0,C 180,E1 29917.713,E2 29917.713} C_VEL
LIN {X 0,Y 640.784,Z 181.324,A -85,B 0,C 180,E1 29914.828,E2 29914.828} C_VEL
LIN {X 0,Y 640.733,Z 181.351,A -85,B 0,C 180,E1 29911.834,E2 29911.834} C_VEL
LIN {X 0,Y 640.758,Z 181.337,A -85,B 0,C 180,E1 29909.135,E2 29909.135} C_VEL
LIN {X 0,Y 640.739,Z 181.342,A -85,B 0,C 180,E1 29906.007,E2 29906.007} C_VEL
LIN {X 0,Y 640.757,Z 181.351,A -85,B 0,C 180,E1 29903.22,E2 29903.22} C_VEL
LIN {X 0,Y 640.739,Z 181.35,A -85,B 0,C 180,E1 29900.064,E2 29900.064} C_VEL
LIN {X 0,Y 640.752,Z 181.346,A -85,B 0,C 180,E1 29897.341,E2 29897.341} C_VEL
LIN {X 0,Y 640.74,Z 181.349,A -85,B 0,C 180,E1 29894.182,E2 29894.182} C_VEL
LIN {X 0,Y 640.75,Z 181.342,A -85,B 0,C 180,E1 29891.431,E2 29891.431} C_VEL
LIN {X 0,Y 640.74,Z 181.344,A -85,B 0,C 180,E1 29888.254,E2 29888.254} C_VEL
LIN {X 0,Y 640.737,Z 181.348,A -85,B 0,C 180,E1 29885.642,E2 29885.642} C_VEL
LIN {X 0,Y 640.756,Z 181.34,A -85,B 0,C 180,E1 29882.504,E2 29882.504} C_VEL
LIN {X 0,Y 640.733,Z 181.35,A -85,B 0,C 180,E1 29879.821,E2 29879.821} C_VEL
LIN {X 0,Y 640.782,Z 181.343,A -85,B 0,C 180,E1 29876.78,E2 29876.78} C_VEL
LIN {X 0,Y 640.731,Z 181.349,A -85,B 0,C 180,E1 29873.998,E2 29873.998} C_VEL
LIN {X 0,Y 640.807,Z 181.343,A -85,B 0,C 180,E1 29871.023,E2 29871.023} C_VEL
LIN {X 0,Y 640.73,Z 181.346,A -85,B 0,C 180,E1 29868.112,E2 29868.112} C_VEL
LIN {X 0,Y 640.823,Z 181.347,A -85,B 0,C 180,E1 29865.173,E2 29865.173} C_VEL
LIN {X 0,Y 640.731,Z 181.342,A -85,B 0,C 180,E1 29862.19,E2 29862.19} C_VEL
LIN {X 0,Y 640.814,Z 181.346,A -85,B 0,C 180,E1 29859.256,E2 29859.256} C_VEL
LIN {X 0,Y 640.732,Z 181.35,A -85,B 0,C 180,E1 29856.336,E2 29856.336} C_VEL
LIN {X 0,Y 640.807,Z 181.33,A -85,B 0,C 180,E1 29853.376,E2 29853.376} C_VEL
LIN {X 0,Y 640.732,Z 181.338,A -85,B 0,C 180,E1 29850.453,E2 29850.453} C_VEL
LIN {X 0,Y 640.77,Z 181.351,A -85,B 0,C 180,E1 29847.741,E2 29847.741} C_VEL
LIN {X 0,Y 640.738,Z 181.34,A -85,B 0,C 180,E1 29844.691,E2 29844.691} C_VEL
LIN {X 0,Y 640.754,Z 181.352,A -85,B 0,C 180,E1 29841.946,E2 29841.946} C_VEL
LIN {X 0,Y 640.741,Z 181.35,A -85,B 0,C 180,E1 29838.77,E2 29838.77} C_VEL
LIN {X 0,Y 640.757,Z 181.343,A -85,B 0,C 180,E1 29835.995,E2 29835.995} C_VEL
LIN {X 0,Y 640.739,Z 181.346,A -85,B 0,C 180,E1 29832.823,E2 29832.823} C_VEL
LIN {X 0,Y 640.751,Z 181.355,A -85,B 0,C 180,E1 29830.12,E2 29830.12} C_VEL
LIN {X 0,Y 640.738,Z 181.314,A -85,B 0,C 180,E1 29826.922,E2 29826.922} C_VEL
LIN {X 0,Y 640.756,Z 181.506,A -85,B 0,C 180,E1 29824.498,E2 29824.498} C_VEL
LIN {X 0,Y 646.698,Z 200.886,A -85,B 0,C 180,E1 29822.337,E2 29822.337} C_VEL
LIN {X 0,Y 648.463,Z 207.835,A -85,B 0,C 180,E1 29821.614,E2 29821.614} C_VEL
LIN {X 0,Y 647.799,Z 225.092,A -85,B 0,C 180,E1 29820.128,E2 29820.128} C_VEL
LIN {X 0,Y 652.986,Z 249.076,A -85,B 0,C 180,E1 29819.563,E2 29819.563} C_VEL
LIN {X 0,Y 650.351,Z 519.06,A -85,B 0,C 180,E1 29816.384,E2 29816.384} C_VEL
LIN {X 0,Y 649.882,Z 539.793,A -85,B 0,C 180,E1 29816.058,E2 29816.058} C_VEL
LIN {X 0,Y 649.377,Z 557.413,A -85,B 0,C 180,E1 29815.67,E2 29815.67} C_VEL
LIN {X 0,Y 648.786,Z 574.205,A -85,B 0,C 180,E1 29815.199,E2 29815.199} C_VEL
LIN {X 0,Y 648.119,Z 590.337,A -85,B 0,C 180,E1 29814.649,E2 29814.649} C_VEL
LIN {X 0,Y 647.389,Z 606.088,A -85,B 0,C 180,E1 29814.011,E2 29814.011} C_VEL
LIN {X 0,Y 646.602,Z 621.823,A -85,B 0,C 180,E1 29813.269,E2 29813.269} C_VEL
LIN {X 0,Y 645.755,Z 637.974,A -85,B 0,C 180,E1 29812.387,E2 29812.387} C_VEL
LIN {X 0,Y 644.738,Z 657.006,A -85,B 0,C 180,E1 29811.18,E2 29811.18} C_VEL
LIN {X 0,Y 643.754,Z 674.156,A -85,B 0,C 180,E1 29809.883,E2 29809.883} C_VEL
LIN {X 0,Y 643.011,Z 687.486,A -85,B 0,C 180,E1 29808.736,E2 29808.736} C_VEL
LIN {X 0,Y 642.365,Z 699.466,A -85,B 0,C 180,E1 29807.574,E2 29807.574} C_VEL
LIN {X 0,Y 641.771,Z 711.183,A -85,B 0,C 180,E1 29806.284,E2 29806.284} C_VEL
LIN {X 0,Y 641.252,Z 722.212,A -85,B 0,C 180,E1 29804.907,E2 29804.907} C_VEL
LIN {X 0,Y 640.78,Z 733.705,A -85,B 0,C 180,E1 29803.259,E2 29803.259} C_VEL
LIN {X 0,Y 640.383,Z 744.785,A -85,B 0,C 180,E1 29801.345,E2 29801.345} C_VEL
LIN {X 0,Y 640.173,Z 752.503,A -85,B 0,C 180,E1 29799.746,E2 29799.746} C_VEL
LIN {X 0,Y 640.051,Z 758.839,A -85,B 0,C 180,E1 29798.172,E2 29798.172} C_VEL
LIN {X 0,Y 639.961,Z 764.126,A -85,B 0,C 180,E1 29796.548,E2 29796.548} C_VEL
LIN {X 0,Y 639.92,Z 768.802,A -85,B 0,C 180,E1 29794.66,E2 29794.66} C_VEL
LIN {X 0,Y 639.911,Z 771.986,A -85,B 0,C 180,E1 29792.597,E2 29792.597} C_VEL
LIN {X 0,Y 639.91,Z 773.265,A -85,B 0,C 180,E1 29790.806,E2 29790.806} C_VEL
LIN {X 0,Y 639.91,Z 773.265,A -85,B 0,C 180,E1 29789.194,E2 29789.194} C_VEL
LIN {X 0,Y 639.911,Z 771.986,A -85,B 0,C 180,E1 29787.403,E2 29787.403} C_VEL
LIN {X 0,Y 639.92,Z 768.802,A -85,B 0,C 180,E1 29785.34,E2 29785.34} C_VEL
LIN {X 0,Y 639.961,Z 764.126,A -85,B 0,C 180,E1 29783.452,E2 29783.452} C_VEL
LIN {X 0,Y 640.051,Z 758.839,A -85,B 0,C 180,E1 29781.828,E2 29781.828} C_VEL
LIN {X 0,Y 640.173,Z 752.503,A -85,B 0,C 180,E1 29780.254,E2 29780.254} C_VEL
LIN {X 0,Y 640.383,Z 744.785,A -85,B 0,C 180,E1 29778.655,E2 29778.655} C_VEL
LIN {X 0,Y 640.78,Z 733.705,A -85,B 0,C 180,E1 29776.741,E2 29776.741} C_VEL
LIN {X 0,Y 641.252,Z 722.212,A -85,B 0,C 180,E1 29775.093,E2 29775.093} C_VEL
LIN {X 0,Y 641.77,Z 711.182,A -85,B 0,C 180,E1 29773.716,E2 29773.716} C_VEL
LIN {X 0,Y 642.365,Z 699.465,A -85,B 0,C 180,E1 29772.426,E2 29772.426} C_VEL
LIN {X 0,Y 643.036,Z 687.079,A -85,B 0,C 180,E1 29771.226,E2 29771.226} C_VEL
LIN {X 0,Y 643.918,Z 671.351,A -85,B 0,C 180,E1 29769.885,E2 29769.885} C_VEL
LIN {X 0,Y 644.95,Z 652.778,A -85,B 0,C 180,E1 29768.541,E2 29768.541} C_VEL
LIN {X 0,Y 645.789,Z 637.242,A -85,B 0,C 180,E1 29767.571,E2 29767.571} C_VEL
LIN {X 0,Y 646.623,Z 621.425,A -85,B 0,C 180,E1 29766.711,E2 29766.711} C_VEL
LIN {X 0,Y 647.389,Z 606.088,A -85,B 0,C 180,E1 29765.989,E2 29765.989} C_VEL
LIN {X 0,Y 648.158,Z 589.426,A -85,B 0,C 180,E1 29765.317,E2 29765.317} C_VEL
LIN {X 0,Y 648.867,Z 572.128,A -85,B 0,C 180,E1 29764.736,E2 29764.736} C_VEL
LIN {X 0,Y 649.617,Z 550.932,A -85,B 0,C 180,E1 29764.167,E2 29764.167} C_VEL
LIN {X 0,Y 650.177,Z 528.3,A -85,B 0,C 180,E1 29763.747,E2 29763.747} C_VEL
LIN {X 0,Y 650.738,Z 478.737,A -85,B 0,C 180,E1 29763.141,E2 29763.141} C_VEL
LIN {X 0,Y 652.877,Z 247.678,A -85,B 0,C 180,E1 29760.414,E2 29760.414} C_VEL
LIN {X 0,Y 647.738,Z 224.416,A -85,B 0,C 180,E1 29759.839,E2 29759.839} C_VEL
LIN {X 0,Y 648.331,Z 206.708,A -85,B 0,C 180,E1 29758.275,E2 29758.275} C_VEL
LIN {X 0,Y 641.323,Z 183.497,A -85,B 0,C 180,E1 29755.753,E2 29755.753} C_VEL
LIN {X 0,Y 640.749,Z 181.471,A -85,B 0,C 180,E1 29755.482,E2 29755.482} C_VEL
LIN {X 0,Y 640.789,Z 181.303,A -85,B 0,C 180,E1 29752.585,E2 29752.585} C_VEL
LIN {X 0,Y 640.735,Z 181.355,A -85,B 0,C 180,E1 29749.601,E2 29749.601} C_VEL
LIN {X 0,Y 640.763,Z 181.345,A -85,B 0,C 180,E1 29746.891,E2 29746.891} C_VEL
LIN {X 0,Y 640.744,Z 181.346,A -85,B 0,C 180,E1 29743.858,E2 29743.858} C_VEL
LIN {X 0,Y 640.752,Z 181.35,A -85,B 0,C 180,E1 29741.095,E2 29741.095} C_VEL
LIN {X 0,Y 640.745,Z 181.352,A -85,B 0,C 180,E1 29737.941,E2 29737.941} C_VEL
LIN {X 0,Y 640.741,Z 181.34,A -85,B 0,C 180,E1 29735.268,E2 29735.268} C_VEL
LIN {X 0,Y 640.749,Z 181.35,A -85,B 0,C 180,E1 29732.044,E2 29732.044} C_VEL
LIN {X 0,Y 640.735,Z 181.338,A -85,B 0,C 180,E1 29729.444,E2 29729.444} C_VEL
LIN {X 0,Y 640.778,Z 181.34,A -85,B 0,C 180,E1 29726.406,E2 29726.406} C_VEL
LIN {X 0,Y 640.733,Z 181.35,A -85,B 0,C 180,E1 29723.645,E2 29723.645} C_VEL
LIN {X 0,Y 640.805,Z 181.348,A -85,B 0,C 180,E1 29720.649,E2 29720.649} C_VEL
LIN {X 0,Y 640.733,Z 181.341,A -85,B 0,C 180,E1 29717.717,E2 29717.717} C_VEL
LIN {X 0,Y 640.801,Z 181.345,A -85,B 0,C 180,E1 29714.693,E2 29714.693} C_VEL
LIN {X 0,Y 640.731,Z 181.346,A -85,B 0,C 180,E1 29711.796,E2 29711.796} C_VEL
LIN {X 0,Y 640.805,Z 181.339,A -85,B 0,C 180,E1 29708.796,E2 29708.796} C_VEL
LIN {X 0,Y 640.731,Z 181.35,A -85,B 0,C 180,E1 29705.912,E2 29705.912} C_VEL
LIN {X 0,Y 640.809,Z 181.339,A -85,B 0,C 180,E1 29702.952,E2 29702.952} C_VEL
LIN {X 0,Y 640.73,Z 181.35,A -85,B 0,C 180,E1 29700,E2 29700} C_VEL
LIN {X 0,Y 640.808,Z 181.34,A -85,B 0,C 180,E1 29697.048,E2 29697.048} C_VEL
LIN {X 0,Y 640.73,Z 181.348,A -85,B 0,C 180,E1 29694.088,E2 29694.088} C_VEL
LIN {X 0,Y 640.804,Z 181.345,A -85,B 0,C 180,E1 29691.204,E2 29691.204} C_VEL
LIN {X 0,Y 640.73,Z 181.343,A -85,B 0,C 180,E1 29688.204,E2 29688.204} C_VEL
LIN {X 0,Y 640.804,Z 181.35,A -85,B 0,C 180,E1 29685.265,E2 29685.265} C_VEL
LIN {X 0,Y 640.732,Z 181.346,A -85,B 0,C 180,E1 29682.284,E2 29682.284} C_VEL
LIN {X 0,Y 640.802,Z 181.346,A -85,B 0,C 180,E1 29679.351,E2 29679.351} C_VEL
LIN {X 0,Y 640.731,Z 181.351,A -85,B 0,C 180,E1 29676.355,E2 29676.355} C_VEL
LIN {X 0,Y 640.788,Z 181.328,A -85,B 0,C 180,E1 29673.495,E2 29673.495} C_VEL
LIN {X 0,Y 640.734,Z 181.343,A -85,B 0,C 180,E1 29670.536,E2 29670.536} C_VEL
LIN {X 0,Y 640.749,Z 181.351,A -85,B 0,C 180,E1 29667.912,E2 29667.912} C_VEL
LIN {X 0,Y 640.737,Z 181.328,A -85,B 0,C 180,E1 29664.732,E2 29664.732} C_VEL
LIN {X 0,Y 640.748,Z 181.35,A -85,B 0,C 180,E1 29661.994,E2 29661.994} C_VEL
LIN {X 0,Y 640.741,Z 181.351,A -85,B 0,C 180,E1 29658.77,E2 29658.77} C_VEL
LIN {X 0,Y 640.755,Z 181.352,A -85,B 0,C 180,E1 29655.996,E2 29655.996} C_VEL
LIN {X 0,Y 640.736,Z 181.352,A -85,B 0,C 180,E1 29654.25,E2 29654.25} C_VEL
LIN {X 0,Y 639.796,Z 181.475,A -85,B 0,C 180,E1 29653.561,E2 29653.561} C_VEL
LIN {X 0,Y 633.3,Z 182.286,A -85,B 0,C 180,E1 29651.58,E2 29651.58} C_VEL
LIN {X 0,Y 632.824,Z 182.34,A -85,B 0,C 180,E1 29651.128,E2 29651.128} C_VEL
LIN {X 0,Y 632.794,Z 182.342,A -85,B 0,C 180,E1 29648.382,E2 29648.382} C_VEL
LIN {X 0,Y 632.841,Z 182.34,A -85,B 0,C 180,E1 29645.324,E2 29645.324} C_VEL
LIN {X 0,Y 632.795,Z 182.342,A -85,B 0,C 180,E1 29642.458,E2 29642.458} C_VEL
LIN {X 0,Y 632.846,Z 182.339,A -85,B 0,C 180,E1 29639.427,E2 29639.427} C_VEL
LIN {X 0,Y 632.794,Z 182.341,A -85,B 0,C 180,E1 29636.559,E2 29636.559} C_VEL
LIN {X 0,Y 632.855,Z 182.34,A -85,B 0,C 180,E1 29633.558,E2 29633.558} C_VEL
LIN {X 0,Y 632.792,Z 182.342,A -85,B 0,C 180,E1 29630.701,E2 29630.701} C_VEL
LIN {X 0,Y 632.859,Z 182.34,A -85,B 0,C 180,E1 29627.657,E2 29627.657} C_VEL
LIN {X 0,Y 632.792,Z 182.343,A -85,B 0,C 180,E1 29624.736,E2 29624.736} C_VEL
LIN {X 0,Y 632.862,Z 182.338,A -85,B 0,C 180,E1 29621.758,E2 29621.758} C_VEL
LIN {X 0,Y 632.791,Z 182.342,A -85,B 0,C 180,E1 29618.815,E2 29618.815} C_VEL
LIN {X 0,Y 632.871,Z 182.337,A -85,B 0,C 180,E1 29615.894,E2 29615.894} C_VEL
LIN {X 0,Y 632.791,Z 182.344,A -85,B 0,C 180,E1 29612.898,E2 29612.898} C_VEL
LIN {X 0,Y 632.868,Z 182.338,A -85,B 0,C 180,E1 29609.91,E2 29609.91} C_VEL
LIN {X 0,Y 632.791,Z 182.344,A -85,B 0,C 180,E1 29606.921,E2 29606.921} C_VEL
LIN {X 0,Y 632.86,Z 182.338,A -85,B 0,C 180,E1 29603.924,E2 29603.924} C_VEL
LIN {X 0,Y 632.792,Z 182.342,A -85,B 0,C 180,E1 29601.093,E2 29601.093} C_VEL
LIN {X 0,Y 632.866,Z 182.339,A -85,B 0,C 180,E1 29598.057,E2 29598.057} C_VEL
LIN {X 0,Y 632.79,Z 182.344,A -85,B 0,C 180,E1 29595.17,E2 29595.17} C_VEL
LIN {X 0,Y 632.869,Z 182.339,A -85,B 0,C 180,E1 29592.249,E2 29592.249} C_VEL
LIN {X 0,Y 632.792,Z 182.342,A -85,B 0,C 180,E1 29589.274,E2 29589.274} C_VEL
LIN {X 0,Y 632.861,Z 182.339,A -85,B 0,C 180,E1 29586.402,E2 29586.402} C_VEL
LIN {X 0,Y 632.794,Z 182.341,A -85,B 0,C 180,E1 29583.425,E2 29583.425} C_VEL
LIN {X 0,Y 632.853,Z 182.339,A -85,B 0,C 180,E1 29580.525,E2 29580.525} C_VEL
LIN {X 0,Y 632.794,Z 182.342,A -85,B 0,C 180,E1 29577.509,E2 29577.509} C_VEL
LIN {X 0,Y 632.85,Z 182.339,A -85,B 0,C 180,E1 29574.614,E2 29574.614} C_VEL
LIN {X 0,Y 632.794,Z 182.342,A -85,B 0,C 180,E1 29571.605,E2 29571.605} C_VEL
LIN {X 0,Y 632.82,Z 182.34,A -85,B 0,C 180,E1 29568.911,E2 29568.911} C_VEL
LIN {X 0,Y 632.802,Z 182.341,A -85,B 0,C 180,E1 29565.835,E2 29565.835} C_VEL
LIN {X 0,Y 632.815,Z 182.341,A -85,B 0,C 180,E1 29563.047,E2 29563.047} C_VEL
LIN {X 0,Y 632.802,Z 182.34,A -85,B 0,C 180,E1 29559.905,E2 29559.905} C_VEL
LIN {X 0,Y 632.803,Z 182.339,A -85,B 0,C 180,E1 29557.226,E2 29557.226} C_VEL
LIN {X 0,Y 632.8,Z 182.331,A -85,B 0,C 180,E1 29553.959,E2 29553.959} C_VEL
LIN {X 0,Y 632.811,Z 182.34,A -85,B 0,C 180,E1 29551.216,E2 29551.216} C_VEL
LIN {X 0,Y 632.804,Z 182.303,A -85,B 0,C 180,E1 29548.091,E2 29548.091} C_VEL
LIN {X 0,Y 632.805,Z 182.331,A -85,B 0,C 180,E1 29545.353,E2 29545.353} C_VEL
LIN {X 0,Y 632.802,Z 182.332,A -85,B 0,C 180,E1 29542.09,E2 29542.09} C_VEL
LIN {X 0,Y 632.809,Z 182.339,A -85,B 0,C 180,E1 29539.379,E2 29539.379} C_VEL
LIN {X 0,Y 632.801,Z 182.336,A -85,B 0,C 180,E1 29536.143,E2 29536.143} C_VEL
LIN {X 0,Y 632.802,Z 182.338,A -85,B 0,C 180,E1 29533.524,E2 29533.524} C_VEL
LIN {X 0,Y 632.806,Z 182.339,A -85,B 0,C 180,E1 29530.285,E2 29530.285} C_VEL
LIN {X 0,Y 632.805,Z 182.333,A -85,B 0,C 180,E1 29527.536,E2 29527.536} C_VEL
LIN {X 0,Y 632.805,Z 182.339,A -85,B 0,C 180,E1 29524.35,E2 29524.35} C_VEL
LIN {X 0,Y 632.803,Z 182.329,A -85,B 0,C 180,E1 29521.63,E2 29521.63} C_VEL
LIN {X 0,Y 632.803,Z 182.334,A -85,B 0,C 180,E1 29518.37,E2 29518.37} C_VEL
LIN {X 0,Y 632.815,Z 182.334,A -85,B 0,C 180,E1 29515.559,E2 29515.559} C_VEL
LIN {X 0,Y 632.804,Z 182.327,A -85,B 0,C 180,E1 29512.464,E2 29512.464} C_VEL
LIN {X 0,Y 632.808,Z 182.338,A -85,B 0,C 180,E1 29509.715,E2 29509.715} C_VEL
LIN {X 0,Y 632.802,Z 182.335,A -85,B 0,C 180,E1 29506.476,E2 29506.476} C_VEL
LIN {X 0,Y 632.804,Z 182.339,A -85,B 0,C 180,E1 29503.853,E2 29503.853} C_VEL
LIN {X 0,Y 632.805,Z 182.34,A -85,B 0,C 180,E1 29500.593,E2 29500.593} C_VEL
LIN {X 0,Y 632.803,Z 182.333,A -85,B 0,C 180,E1 29497.91,E2 29497.91} C_VEL
LIN {X 0,Y 632.806,Z 182.335,A -85,B 0,C 180,E1 29494.646,E2 29494.646} C_VEL
LIN {X 0,Y 632.814,Z 182.309,A -85,B 0,C 180,E1 29491.831,E2 29491.831} C_VEL
LIN {X 0,Y 632.802,Z 182.34,A -85,B 0,C 180,E1 29488.677,E2 29488.677} C_VEL
LIN {X 0,Y 632.807,Z 182.334,A -85,B 0,C 180,E1 29485.989,E2 29485.989} C_VEL
LIN {X 0,Y 632.804,Z 182.341,A -85,B 0,C 180,E1 29482.758,E2 29482.758} C_VEL
LIN {X 0,Y 632.804,Z 182.328,A -85,B 0,C 180,E1 29480.095,E2 29480.095} C_VEL
LIN {X 0,Y 632.804,Z 182.335,A -85,B 0,C 180,E1 29476.828,E2 29476.828} C_VEL
LIN {X 0,Y 632.816,Z 182.34,A -85,B 0,C 180,E1 29474.033,E2 29474.033} C_VEL
LIN {X 0,Y 632.804,Z 182.344,A -85,B 0,C 180,E1 29470.849,E2 29470.849} C_VEL
LIN {X 0,Y 632.806,Z 182.299,A -85,B 0,C 180,E1 29468.151,E2 29468.151} C_VEL
LIN {X 0,Y 632.81,Z 182.361,A -85,B 0,C 180,E1 29464.994,E2 29464.994} C_VEL
LIN {X 0,Y 632.868,Z 182.791,A -85,B 0,C 180,E1 29464.825,E2 29464.825} C_VEL
LIN {X 0,Y 639.184,Z 203.249,A -85,B 0,C 180,E1 29462.523,E2 29462.523} C_VEL
LIN {X 0,Y 641.043,Z 210.265,A -85,B 0,C 180,E1 29461.779,E2 29461.779} C_VEL
LIN {X 0,Y 640.445,Z 224.835,A -85,B 0,C 180,E1 29460.512,E2 29460.512} C_VEL
LIN {X 0,Y 646.001,Z 250.565,A -85,B 0,C 180,E1 29459.894,E2 29459.894} C_VEL
LIN {X 0,Y 643.161,Z 519.611,A -85,B 0,C 180,E1 29456.691,E2 29456.691} C_VEL
LIN {X 0,Y 642.671,Z 539.78,A -85,B 0,C 180,E1 29456.37,E2 29456.37} C_VEL
LIN {X 0,Y 642.123,Z 557.466,A -85,B 0,C 180,E1 29455.976,E2 29455.976} C_VEL
LIN {X 0,Y 641.51,Z 573.709,A -85,B 0,C 180,E1 29455.516,E2 29455.516} C_VEL
LIN {X 0,Y 640.793,Z 589.872,A -85,B 0,C 180,E1 29454.961,E2 29454.961} C_VEL
LIN {X 0,Y 640,Z 605.911,A -85,B 0,C 180,E1 29454.306,E2 29454.306} C_VEL
LIN {X 0,Y 639.205,Z 620.726,A -85,B 0,C 180,E1 29453.603,E2 29453.603} C_VEL
LIN {X 0,Y 638.322,Z 636.182,A -85,B 0,C 180,E1 29452.759,E2 29452.759} C_VEL
LIN {X 0,Y 637.44,Z 651.177,A -85,B 0,C 180,E1 29451.821,E2 29451.821} C_VEL
LIN {X 0,Y 636.47,Z 667.556,A -85,B 0,C 180,E1 29450.649,E2 29450.649} C_VEL
LIN {X 0,Y 635.393,Z 685.401,A -85,B 0,C 180,E1 29449.151,E2 29449.151} C_VEL
LIN {X 0,Y 634.627,Z 698.409,A -85,B 0,C 180,E1 29447.89,E2 29447.89} C_VEL
LIN {X 0,Y 633.98,Z 710.302,A -85,B 0,C 180,E1 29446.584,E2 29446.584} C_VEL
LIN {X 0,Y 633.447,Z 720.798,A -85,B 0,C 180,E1 29445.282,E2 29445.282} C_VEL
LIN {X 0,Y 633.009,Z 730.014,A -85,B 0,C 180,E1 29443.984,E2 29443.984} C_VEL
LIN {X 0,Y 632.661,Z 738.661,A -85,B 0,C 180,E1 29442.596,E2 29442.596} C_VEL
LIN {X 0,Y 632.369,Z 746.638,A -85,B 0,C 180,E1 29441.121,E2 29441.121} C_VEL
LIN {X 0,Y 632.163,Z 753.84,A -85,B 0,C 180,E1 29439.559,E2 29439.559} C_VEL
LIN {X 0,Y 632.015,Z 761.132,A -85,B 0,C 180,E1 29437.636,E2 29437.636} C_VEL
LIN {X 0,Y 631.944,Z 766.823,A -85,B 0,C 180,E1 29435.594,E2 29435.594} C_VEL
LIN {X 0,Y 631.923,Z 770.213,A -85,B 0,C 180,E1 29433.901,E2 29433.901} C_VEL
LIN {X 0,Y 631.91,Z 772.329,A -85,B 0,C 180,E1 29432.267,E2 29432.267} C_VEL
LIN {X 0,Y 631.904,Z 773.318,A -85,B 0,C 180,E1 29430.635,E2 29430.635} C_VEL
LIN {X 0,Y 631.904,Z 773.174,A -85,B 0,C 180,E1 29428.912,E2 29428.912} C_VEL
LIN {X 0,Y 631.904,Z 771.38,A -85,B 0,C 180,E1 29426.826,E2 29426.826} C_VEL
LIN {X 0,Y 631.921,Z 767.978,A -85,B 0,C 180,E1 29424.917,E2 29424.917} C_VEL
LIN {X 0,Y 631.967,Z 763.853,A -85,B 0,C 180,E1 29423.277,E2 29423.277} C_VEL
LIN {X 0,Y 632.063,Z 758.833,A -85,B 0,C 180,E1 29421.724,E2 29421.724} C_VEL
LIN {X 0,Y 632.197,Z 752.654,A -85,B 0,C 180,E1 29420.166,E2 29420.166} C_VEL
LIN {X 0,Y 632.416,Z 745.222,A -85,B 0,C 180,E1 29418.598,E2 29418.598} C_VEL
LIN {X 0,Y 632.824,Z 734.748,A -85,B 0,C 180,E1 29416.733,E2 29416.733} C_VEL
LIN {X 0,Y 633.349,Z 722.902,A -85,B 0,C 180,E1 29414.997,E2 29414.997} C_VEL
LIN {X 0,Y 633.894,Z 711.885,A -85,B 0,C 180,E1 29413.602,E2 29413.602} C_VEL
LIN {X 0,Y 634.522,Z 700.189,A -85,B 0,C 180,E1 29412.297,E2 29412.297} C_VEL
LIN {X 0,Y 635.271,Z 687.4,A -85,B 0,C 180,E1 29411.036,E2 29411.036} C_VEL
LIN {X 0,Y 636.072,Z 673.978,A -85,B 0,C 180,E1 29409.866,E2 29409.866} C_VEL
LIN {X 0,Y 637.166,Z 656.422,A -85,B 0,C 180,E1 29408.526,E2 29408.526} C_VEL
LIN {X 0,Y 638.234,Z 637.769,A -85,B 0,C 180,E1 29407.333,E2 29407.333} C_VEL
LIN {X 0,Y 639.136,Z 621.927,A -85,B 0,C 180,E1 29406.458,E2 29406.458} C_VEL
LIN {X 0,Y 639.943,Z 606.974,A -85,B 0,C 180,E1 29405.74,E2 29405.74} C_VEL
LIN {X 0,Y 640.737,Z 591.072,A -85,B 0,C 180,E1 29405.084,E2 29405.084} C_VEL
LIN {X 0,Y 641.461,Z 574.926,A -85,B 0,C 180,E1 29404.522,E2 29404.522} C_VEL
LIN {X 0,Y 642.111,Z 557.809,A -85,B 0,C 180,E1 29404.033,E2 29404.033} C_VEL
LIN {X 0,Y 642.655,Z 540.356,A -85,B 0,C 180,E1 29403.642,E2 29403.642} C_VEL
LIN {X 0,Y 643.115,Z 521.527,A -85,B 0,C 180,E1 29403.336,E2 29403.336} C_VEL
LIN {X 0,Y 645.929,Z 257.183,A -85,B 0,C 180,E1 29400.185,E2 29400.185} C_VEL
LIN {X 0,Y 645.803,Z 248.742,A -85,B 0,C 180,E1 29400.073,E2 29400.073} C_VEL
LIN {X 0,Y 640.425,Z 224.659,A -85,B 0,C 180,E1 29399.48,E2 29399.48} C_VEL
LIN {X 0,Y 640.964,Z 209.555,A -85,B 0,C 180,E1 29398.148,E2 29398.148} C_VEL
LIN {X 0,Y 634.278,Z 187.231,A -85,B 0,C 180,E1 29395.695,E2 29395.695} C_VEL
LIN {X 0,Y 632.821,Z 182.487,A -85,B 0,C 180,E1 29395.117,E2 29395.117} C_VEL
LIN {X 0,Y 632.824,Z 182.295,A -85,B 0,C 180,E1 29392.041,E2 29392.041} C_VEL
LIN {X 0,Y 632.796,Z 182.344,A -85,B 0,C 180,E1 29389.329,E2 29389.329} C_VEL
LIN {X 0,Y 632.863,Z 182.34,A -85,B 0,C 180,E1 29386.343,E2 29386.343} C_VEL
LIN {X 0,Y 632.794,Z 182.335,A -85,B 0,C 180,E1 29383.385,E2 29383.385} C_VEL
LIN {X 0,Y 632.856,Z 182.323,A -85,B 0,C 180,E1 29380.375,E2 29380.375} C_VEL
LIN {X 0,Y 632.794,Z 182.341,A -85,B 0,C 180,E1 29377.523,E2 29377.523} C_VEL
LIN {X 0,Y 632.87,Z 182.319,A -85,B 0,C 180,E1 29374.555,E2 29374.555} C_VEL
LIN {X 0,Y 632.795,Z 182.339,A -85,B 0,C 180,E1 29371.618,E2 29371.618} C_VEL
LIN {X 0,Y 632.874,Z 182.304,A -85,B 0,C 180,E1 29368.705,E2 29368.705} C_VEL
LIN {X 0,Y 632.794,Z 182.335,A -85,B 0,C 180,E1 29365.756,E2 29365.756} C_VEL
LIN {X 0,Y 632.877,Z 182.33,A -85,B 0,C 180,E1 29362.773,E2 29362.773} C_VEL
LIN {X 0,Y 632.791,Z 182.339,A -85,B 0,C 180,E1 29359.764,E2 29359.764} C_VEL
LIN {X 0,Y 632.871,Z 182.328,A -85,B 0,C 180,E1 29356.803,E2 29356.803} C_VEL
LIN {X 0,Y 632.793,Z 182.334,A -85,B 0,C 180,E1 29353.897,E2 29353.897} C_VEL
LIN {X 0,Y 632.867,Z 182.335,A -85,B 0,C 180,E1 29350.929,E2 29350.929} C_VEL
LIN {X 0,Y 632.793,Z 182.328,A -85,B 0,C 180,E1 29347.993,E2 29347.993} C_VEL
LIN {X 0,Y 632.847,Z 182.339,A -85,B 0,C 180,E1 29345.167,E2 29345.167} C_VEL
LIN {X 0,Y 632.795,Z 182.335,A -85,B 0,C 180,E1 29342.173,E2 29342.173} C_VEL
LIN {X 0,Y 632.819,Z 182.339,A -85,B 0,C 180,E1 29339.457,E2 29339.457} C_VEL
LIN {X 0,Y 632.796,Z 182.339,A -85,B 0,C 180,E1 29336.286,E2 29336.286} C_VEL
LIN {X 0,Y 632.826,Z 182.336,A -85,B 0,C 180,E1 29333.468,E2 29333.468} C_VEL
LIN {X 0,Y 632.799,Z 182.339,A -85,B 0,C 180,E1 29330.35,E2 29330.35} C_VEL
LIN {X 0,Y 632.828,Z 182.33,A -85,B 0,C 180,E1 29327.499,E2 29327.499} C_VEL
LIN {X 0,Y 632.796,Z 182.337,A -85,B 0,C 180,E1 29324.418,E2 29324.418} C_VEL
LIN {X 0,Y 632.817,Z 182.335,A -85,B 0,C 180,E1 29321.673,E2 29321.673} C_VEL
LIN {X 0,Y 632.8,Z 182.332,A -85,B 0,C 180,E1 29318.521,E2 29318.521} C_VEL
LIN {X 0,Y 632.809,Z 182.34,A -85,B 0,C 180,E1 29315.843,E2 29315.843} C_VEL
LIN {X 0,Y 632.798,Z 182.305,A -85,B 0,C 180,E1 29312.611,E2 29312.611} C_VEL
LIN {X 0,Y 632.806,Z 182.331,A -85,B 0,C 180,E1 29309.941,E2 29309.941} C_VEL
LIN {X 0,Y 632.801,Z 182.331,A -85,B 0,C 180,E1 29306.695,E2 29306.695} C_VEL
LIN {X 0,Y 632.813,Z 182.318,A -85,B 0,C 180,E1 29303.888,E2 29303.888} C_VEL
LIN {X 0,Y 632.8,Z 182.34,A -85,B 0,C 180,E1 29300.728,E2 29300.728} C_VEL
LIN {X 0,Y 632.807,Z 182.34,A -85,B 0,C 180,E1 29298.058,E2 29298.058} C_VEL
LIN {X 0,Y 632.808,Z 182.341,A -85,B 0,C 180,E1 29294.927,E2 29294.927} C_VEL
LIN {X 0,Y 632.804,Z 182.341,A -85,B 0,C 180,E1 29292.178,E2 29292.178} C_VEL
LIN {X 0,Y 632.824,Z 182.34,A -85,B 0,C 180,E1 29291.128,E2 29291.128} C_VEL
LIN {X 0,Y 631.776,Z 182.47,A -85,B 0,C 180,E1 29290.43,E2 29290.43} C_VEL
LIN {X 0,Y 625.37,Z 183.268,A -85,B 0,C 180,E1 29288.474,E2 29288.474} C_VEL
LIN {X 0,Y 624.887,Z 183.331,A -85,B 0,C 180,E1 29287.966,E2 29287.966} C_VEL
LIN {X 0,Y 624.857,Z 183.331,A -85,B 0,C 180,E1 29284.825,E2 29284.825} C_VEL
LIN {X 0,Y 624.896,Z 183.329,A -85,B 0,C 180,E1 29281.976,E2 29281.976} C_VEL
LIN {X 0,Y 624.858,Z 183.331,A -85,B 0,C 180,E1 29278.894,E2 29278.894} C_VEL
LIN {X 0,Y 624.901,Z 183.329,A -85,B 0,C 180,E1 29275.999,E2 29275.999} C_VEL
LIN {X 0,Y 624.86,Z 183.331,A -85,B 0,C 180,E1 29272.979,E2 29272.979} C_VEL
LIN {X 0,Y 624.883,Z 183.331,A -85,B 0,C 180,E1 29270.217,E2 29270.217} C_VEL
LIN {X 0,Y 624.863,Z 183.331,A -85,B 0,C 180,E1 29267.121,E2 29267.121} C_VEL
LIN {X 0,Y 624.874,Z 183.332,A -85,B 0,C 180,E1 29264.359,E2 29264.359} C_VEL
LIN {X 0,Y 624.861,Z 183.333,A -85,B 0,C 180,E1 29261.163,E2 29261.163} C_VEL
LIN {X 0,Y 624.879,Z 183.33,A -85,B 0,C 180,E1 29258.372,E2 29258.372} C_VEL
LIN {X 0,Y 624.861,Z 183.332,A -85,B 0,C 180,E1 29255.233,E2 29255.233} C_VEL
LIN {X 0,Y 624.884,Z 183.333,A -85,B 0,C 180,E1 29252.384,E2 29252.384} C_VEL
LIN {X 0,Y 624.859,Z 183.332,A -85,B 0,C 180,E1 29249.267,E2 29249.267} C_VEL
LIN {X 0,Y 624.886,Z 183.33,A -85,B 0,C 180,E1 29246.423,E2 29246.423} C_VEL
LIN {X 0,Y 624.857,Z 183.333,A -85,B 0,C 180,E1 29243.293,E2 29243.293} C_VEL
LIN {X 0,Y 624.884,Z 183.331,A -85,B 0,C 180,E1 29240.515,E2 29240.515} C_VEL
LIN {X 0,Y 624.859,Z 183.33,A -85,B 0,C 180,E1 29237.432,E2 29237.432} C_VEL
LIN {X 0,Y 624.874,Z 183.333,A -85,B 0,C 180,E1 29234.693,E2 29234.693} C_VEL
LIN {X 0,Y 624.864,Z 183.332,A -85,B 0,C 180,E1 29231.531,E2 29231.531} C_VEL
LIN {X 0,Y 624.871,Z 183.331,A -85,B 0,C 180,E1 29228.802,E2 29228.802} C_VEL
LIN {X 0,Y 624.862,Z 183.332,A -85,B 0,C 180,E1 29225.575,E2 29225.575} C_VEL
LIN {X 0,Y 624.881,Z 183.33,A -85,B 0,C 180,E1 29222.769,E2 29222.769} C_VEL
LIN {X 0,Y 624.859,Z 183.33,A -85,B 0,C 180,E1 29219.599,E2 29219.599} C_VEL
LIN {X 0,Y 624.883,Z 183.331,A -85,B 0,C 180,E1 29216.811,E2 29216.811} C_VEL
LIN {X 0,Y 624.863,Z 183.329,A -85,B 0,C 180,E1 29213.702,E2 29213.702} C_VEL
LIN {X 0,Y 624.879,Z 183.331,A -85,B 0,C 180,E1 29210.902,E2 29210.902} C_VEL
LIN {X 0,Y 624.863,Z 183.33,A -85,B 0,C 180,E1 29207.78,E2 29207.78} C_VEL
LIN {X 0,Y 624.877,Z 183.33,A -85,B 0,C 180,E1 29204.995,E2 29204.995} C_VEL
LIN {X 0,Y 624.863,Z 183.329,A -85,B 0,C 180,E1 29201.857,E2 29201.857} C_VEL
LIN {X 0,Y 624.866,Z 183.329,A -85,B 0,C 180,E1 29199.203,E2 29199.203} C_VEL
LIN {X 0,Y 624.861,Z 183.306,A -85,B 0,C 180,E1 29195.945,E2 29195.945} C_VEL
LIN {X 0,Y 624.872,Z 183.319,A -85,B 0,C 180,E1 29193.179,E2 29193.179} C_VEL
LIN {X 0,Y 624.866,Z 183.32,A -85,B 0,C 180,E1 29190.052,E2 29190.052} C_VEL
LIN {X 0,Y 624.863,Z 183.29,A -85,B 0,C 180,E1 29187.339,E2 29187.339} C_VEL
LIN {X 0,Y 624.864,Z 183.329,A -85,B 0,C 180,E1 29184.082,E2 29184.082} C_VEL
LIN {X 0,Y 624.868,Z 183.321,A -85,B 0,C 180,E1 29181.383,E2 29181.383} C_VEL
LIN {X 0,Y 624.863,Z 183.324,A -85,B 0,C 180,E1 29178.126,E2 29178.126} C_VEL
LIN {X 0,Y 624.877,Z 183.325,A -85,B 0,C 180,E1 29175.309,E2 29175.309} C_VEL
LIN {X 0,Y 624.861,Z 183.319,A -85,B 0,C 180,E1 29172.157,E2 29172.157} C_VEL
LIN {X 0,Y 624.887,Z 183.328,A -85,B 0,C 180,E1 29169.3,E2 29169.3} C_VEL
LIN {X 0,Y 624.861,Z 183.326,A -85,B 0,C 180,E1 29166.247,E2 29166.247} C_VEL
LIN {X 0,Y 624.875,Z 183.327,A -85,B 0,C 180,E1 29163.486,E2 29163.486} C_VEL
LIN {X 0,Y 624.86,Z 183.328,A -85,B 0,C 180,E1 29160.275,E2 29160.275} C_VEL
LIN {X 0,Y 624.878,Z 183.323,A -85,B 0,C 180,E1 29157.524,E2 29157.524} C_VEL
LIN {X 0,Y 624.862,Z 183.327,A -85,B 0,C 180,E1 29154.368,E2 29154.368} C_VEL
LIN {X 0,Y 624.865,Z 183.315,A -85,B 0,C 180,E1 29151.72,E2 29151.72} C_VEL
LIN {X 0,Y 624.863,Z 183.323,A -85,B 0,C 180,E1 29148.462,E2 29148.462} C_VEL
LIN {X 0,Y 624.88,Z 183.324,A -85,B 0,C 180,E1 29145.639,E2 29145.639} C_VEL
LIN {X 0,Y 624.861,Z 183.319,A -85,B 0,C 180,E1 29142.473,E2 29142.473} C_VEL
LIN {X 0,Y 624.894,Z 183.329,A -85,B 0,C 180,E1 29139.585,E2 29139.585} C_VEL
LIN {X 0,Y 624.861,Z 183.328,A -85,B 0,C 180,E1 29136.519,E2 29136.519} C_VEL
LIN {X 0,Y 624.896,Z 183.316,A -85,B 0,C 180,E1 29133.628,E2 29133.628} C_VEL
LIN {X 0,Y 624.858,Z 183.314,A -85,B 0,C 180,E1 29130.577,E2 29130.577} C_VEL
LIN {X 0,Y 624.886,Z 183.329,A -85,B 0,C 180,E1 29127.802,E2 29127.802} C_VEL
LIN {X 0,Y 624.861,Z 183.316,A -85,B 0,C 180,E1 29124.684,E2 29124.684} C_VEL
LIN {X 0,Y 624.886,Z 183.33,A -85,B 0,C 180,E1 29121.855,E2 29121.855} C_VEL
LIN {X 0,Y 624.863,Z 183.328,A -85,B 0,C 180,E1 29118.755,E2 29118.755} C_VEL
LIN {X 0,Y 624.889,Z 183.317,A -85,B 0,C 180,E1 29115.889,E2 29115.889} C_VEL
LIN {X 0,Y 624.863,Z 183.323,A -85,B 0,C 180,E1 29112.842,E2 29112.842} C_VEL
LIN {X 0,Y 624.875,Z 183.334,A -85,B 0,C 180,E1 29110.104,E2 29110.104} C_VEL
LIN {X 0,Y 624.858,Z 183.286,A -85,B 0,C 180,E1 29106.869,E2 29106.869} C_VEL
LIN {X 0,Y 624.923,Z 183.544,A -85,B 0,C 180,E1 29105.246,E2 29105.246} C_VEL
LIN {X 0,Y 630.832,Z 202.866,A -85,B 0,C 180,E1 29103.019,E2 29103.019} C_VEL
LIN {X 0,Y 633.596,Z 213.3,A -85,B 0,C 180,E1 29101.893,E2 29101.893} C_VEL
LIN {X 0,Y 633.053,Z 224.005,A -85,B 0,C 180,E1 29100.934,E2 29100.934} C_VEL
LIN {X 0,Y 639.038,Z 252.027,A -85,B 0,C 180,E1 29100.233,E2 29100.233} C_VEL
LIN {X 0,Y 635.995,Z 519.941,A -85,B 0,C 180,E1 29097.008,E2 29097.008} C_VEL
LIN {X 0,Y 635.483,Z 539.766,A -85,B 0,C 180,E1 29096.688,E2 29096.688} C_VEL
LIN {X 0,Y 634.889,Z 557.405,A -85,B 0,C 180,E1 29096.291,E2 29096.291} C_VEL
LIN {X 0,Y 634.217,Z 574.108,A -85,B 0,C 180,E1 29095.812,E2 29095.812} C_VEL
LIN {X 0,Y 633.444,Z 590.314,A -85,B 0,C 180,E1 29095.246,E2 29095.246} C_VEL
LIN {X 0,Y 632.569,Z 606.797,A -85,B 0,C 180,E1 29094.561,E2 29094.561} C_VEL
LIN {X 0,Y 631.616,Z 623.219,A -85,B 0,C 180,E1 29093.76,E2 29093.76} C_VEL
LIN {X 0,Y 630.421,Z 643.174,A -85,B 0,C 180,E1 29092.617,E2 29092.617} C_VEL
LIN {X 0,Y 629.272,Z 660.438,A -85,B 0,C 180,E1 29091.433,E2 29091.433} C_VEL
LIN {X 0,Y 628.328,Z 674.921,A -85,B 0,C 180,E1 29090.296,E2 29090.296} C_VEL
LIN {X 0,Y 627.508,Z 687.721,A -85,B 0,C 180,E1 29089.16,E2 29089.16} C_VEL
LIN {X 0,Y 626.735,Z 700.011,A -85,B 0,C 180,E1 29087.931,E2 29087.931} C_VEL
LIN {X 0,Y 626.101,Z 710.915,A -85,B 0,C 180,E1 29086.704,E2 29086.704} C_VEL
LIN {X 0,Y 625.499,Z 722.023,A -85,B 0,C 180,E1 29085.291,E2 29085.291} C_VEL
LIN {X 0,Y 624.974,Z 732.981,A -85,B 0,C 180,E1 29083.695,E2 29083.695} C_VEL
LIN {X 0,Y 624.508,Z 744.307,A -85,B 0,C 180,E1 29081.731,E2 29081.731} C_VEL
LIN {X 0,Y 624.244,Z 752.253,A -85,B 0,C 180,E1 29080.054,E2 29080.054} C_VEL
LIN {X 0,Y 624.075,Z 758.496,A -85,B 0,C 180,E1 29078.475,E2 29078.475} C_VEL
LIN {X 0,Y 623.975,Z 763.581,A -85,B 0,C 180,E1 29076.902,E2 29076.902} C_VEL
LIN {X 0,Y 623.935,Z 767.564,A -85,B 0,C 180,E1 29075.332,E2 29075.332} C_VEL
LIN {X 0,Y 623.919,Z 770.646,A -85,B 0,C 180,E1 29073.675,E2 29073.675} C_VEL
LIN {X 0,Y 623.911,Z 772.846,A -85,B 0,C 180,E1 29071.745,E2 29071.745} C_VEL
LIN {X 0,Y 623.901,Z 773.401,A -85,B 0,C 180,E1 29069.633,E2 29069.633} C_VEL
LIN {X 0,Y 623.913,Z 772.497,A -85,B 0,C 180,E1 29067.888,E2 29067.888} C_VEL
LIN {X 0,Y 623.922,Z 770.5,A -85,B 0,C 180,E1 29066.233,E2 29066.233} C_VEL
LIN {X 0,Y 623.935,Z 767.564,A -85,B 0,C 180,E1 29064.667,E2 29064.667} C_VEL
LIN {X 0,Y 623.975,Z 763.581,A -85,B 0,C 180,E1 29063.098,E2 29063.098} C_VEL
LIN {X 0,Y 624.075,Z 758.496,A -85,B 0,C 180,E1 29061.525,E2 29061.525} C_VEL
LIN {X 0,Y 624.244,Z 752.253,A -85,B 0,C 180,E1 29059.946,E2 29059.946} C_VEL
LIN {X 0,Y 624.508,Z 744.307,A -85,B 0,C 180,E1 29058.269,E2 29058.269} C_VEL
LIN {X 0,Y 624.996,Z 732.362,A -85,B 0,C 180,E1 29056.211,E2 29056.211} C_VEL
LIN {X 0,Y 625.499,Z 722.023,A -85,B 0,C 180,E1 29054.709,E2 29054.709} C_VEL
LIN {X 0,Y 626.101,Z 710.915,A -85,B 0,C 180,E1 29053.296,E2 29053.296} C_VEL
LIN {X 0,Y 626.735,Z 700.011,A -85,B 0,C 180,E1 29052.069,E2 29052.069} C_VEL
LIN {X 0,Y 627.54,Z 687.221,A -85,B 0,C 180,E1 29050.793,E2 29050.793} C_VEL
LIN {X 0,Y 628.421,Z 673.475,A -85,B 0,C 180,E1 29049.582,E2 29049.582} C_VEL
LIN {X 0,Y 629.638,Z 655.268,A -85,B 0,C 180,E1 29048.189,E2 29048.189} C_VEL
LIN {X 0,Y 630.73,Z 637.617,A -85,B 0,C 180,E1 29047.05,E2 29047.05} C_VEL
LIN {X 0,Y 631.665,Z 622.39,A -85,B 0,C 180,E1 29046.197,E2 29046.197} C_VEL
LIN {X 0,Y 632.569,Z 606.797,A -85,B 0,C 180,E1 29045.439,E2 29045.439} C_VEL
LIN {X 0,Y 633.443,Z 590.315,A -85,B 0,C 180,E1 29044.754,E2 29044.754} C_VEL
LIN {X 0,Y 634.217,Z 574.107,A -85,B 0,C 180,E1 29044.188,E2 29044.188} C_VEL
LIN {X 0,Y 634.909,Z 556.832,A -85,B 0,C 180,E1 29043.694,E2 29043.694} C_VEL
LIN {X 0,Y 635.521,Z 538.661,A -85,B 0,C 180,E1 29043.29,E2 29043.29} C_VEL
LIN {X 0,Y 636.084,Z 515.451,A -85,B 0,C 180,E1 29042.931,E2 29042.931} C_VEL
LIN {X 0,Y 639.047,Z 251.149,A -85,B 0,C 180,E1 29039.756,E2 29039.756} C_VEL
LIN {X 0,Y 633.056,Z 224.017,A -85,B 0,C 180,E1 29039.066,E2 29039.066} C_VEL
LIN {X 0,Y 633.479,Z 212.003,A -85,B 0,C 180,E1 29037.976,E2 29037.976} C_VEL
LIN {X 0,Y 626.936,Z 190.177,A -85,B 0,C 180,E1 29035.544,E2 29035.544} C_VEL
LIN {X 0,Y 624.912,Z 183.449,A -85,B 0,C 180,E1 29034.722,E2 29034.722} C_VEL
LIN {X 0,Y 624.855,Z 183.29,A -85,B 0,C 180,E1 29031.626,E2 29031.626} C_VEL
LIN {X 0,Y 624.884,Z 183.33,A -85,B 0,C 180,E1 29028.886,E2 29028.886} C_VEL
LIN {X 0,Y 624.863,Z 183.329,A -85,B 0,C 180,E1 29025.767,E2 29025.767} C_VEL
LIN {X 0,Y 624.881,Z 183.324,A -85,B 0,C 180,E1 29022.973,E2 29022.973} C_VEL
LIN {X 0,Y 624.86,Z 183.317,A -85,B 0,C 180,E1 29019.798,E2 29019.798} C_VEL
LIN {X 0,Y 624.883,Z 183.33,A -85,B 0,C 180,E1 29017.027,E2 29017.027} C_VEL
LIN {X 0,Y 624.859,Z 183.323,A -85,B 0,C 180,E1 29013.839,E2 29013.839} C_VEL
LIN {X 0,Y 624.899,Z 183.328,A -85,B 0,C 180,E1 29010.96,E2 29010.96} C_VEL
LIN {X 0,Y 624.86,Z 183.299,A -85,B 0,C 180,E1 29007.96,E2 29007.96} C_VEL
LIN {X 0,Y 624.891,Z 183.323,A -85,B 0,C 180,E1 29005.089,E2 29005.089} C_VEL
LIN {X 0,Y 624.859,Z 183.32,A -85,B 0,C 180,E1 29001.99,E2 29001.99} C_VEL
LIN {X 0,Y 624.89,Z 183.327,A -85,B 0,C 180,E1 28999.149,E2 28999.149} C_VEL
LIN {X 0,Y 624.861,Z 183.326,A -85,B 0,C 180,E1 28996.071,E2 28996.071} C_VEL
LIN {X 0,Y 624.871,Z 183.323,A -85,B 0,C 180,E1 28993.404,E2 28993.404} C_VEL
LIN {X 0,Y 624.865,Z 183.327,A -85,B 0,C 180,E1 28990.231,E2 28990.231} C_VEL
LIN {X 0,Y 624.872,Z 183.317,A -85,B 0,C 180,E1 28987.447,E2 28987.447} C_VEL
LIN {X 0,Y 624.861,Z 183.324,A -85,B 0,C 180,E1 28984.221,E2 28984.221} C_VEL
LIN {X 0,Y 624.887,Z 183.323,A -85,B 0,C 180,E1 28981.375,E2 28981.375} C_VEL
LIN {X 0,Y 624.857,Z 183.318,A -85,B 0,C 180,E1 28978.258,E2 28978.258} C_VEL
LIN {X 0,Y 624.895,Z 183.327,A -85,B 0,C 180,E1 28975.358,E2 28975.358} C_VEL
LIN {X 0,Y 624.857,Z 183.322,A -85,B 0,C 180,E1 28972.275,E2 28972.275} C_VEL
LIN {X 0,Y 624.902,Z 183.328,A -85,B 0,C 180,E1 28969.397,E2 28969.397} C_VEL
LIN {X 0,Y 624.855,Z 183.327,A -85,B 0,C 180,E1 28966.301,E2 28966.301} C_VEL
LIN {X 0,Y 624.89,Z 183.325,A -85,B 0,C 180,E1 28963.548,E2 28963.548} C_VEL
LIN {X 0,Y 624.859,Z 183.328,A -85,B 0,C 180,E1 28960.455,E2 28960.455} C_VEL
LIN {X 0,Y 624.889,Z 183.321,A -85,B 0,C 180,E1 28957.615,E2 28957.615} C_VEL
LIN {X 0,Y 624.859,Z 183.319,A -85,B 0,C 180,E1 28954.504,E2 28954.504} C_VEL
LIN {X 0,Y 624.895,Z 183.291,A -85,B 0,C 180,E1 28951.626,E2 28951.626} C_VEL
LIN {X 0,Y 624.858,Z 183.33,A -85,B 0,C 180,E1 28948.556,E2 28948.556} C_VEL
LIN {X 0,Y 624.891,Z 183.307,A -85,B 0,C 180,E1 28945.72,E2 28945.72} C_VEL
LIN {X 0,Y 624.858,Z 183.328,A -85,B 0,C 180,E1 28942.665,E2 28942.665} C_VEL
LIN {X 0,Y 624.874,Z 183.329,A -85,B 0,C 180,E1 28939.965,E2 28939.965} C_VEL
LIN {X 0,Y 624.862,Z 183.33,A -85,B 0,C 180,E1 28936.774,E2 28936.774} C_VEL
LIN {X 0,Y 624.882,Z 183.33,A -85,B 0,C 180,E1 28933.941,E2 28933.941} C_VEL
LIN {X 0,Y 624.862,Z 183.329,A -85,B 0,C 180,E1 28930.809,E2 28930.809} C_VEL
LIN {X 0,Y 624.877,Z 183.331,A -85,B 0,C 180,E1 28928.069,E2 28928.069} C_VEL
LIN {X 0,Y 624.887,Z 183.331,A -85,B 0,C 180,E1 28927.966,E2 28927.966} C_VEL
LIN {X 0,Y 623.949,Z 183.452,A -85,B 0,C 180,E1 28927.259,E2 28927.259} C_VEL
LIN {X 0,Y 617.469,Z 184.255,A -85,B 0,C 180,E1 28925.279,E2 28925.279} C_VEL
LIN {X 0,Y 616.917,Z 184.32,A -85,B 0,C 180,E1 28924.763,E2 28924.763} C_VEL
LIN {X 0,Y 616.983,Z 184.316,A -85,B 0,C 180,E1 28921.778,E2 28921.778} C_VEL
LIN {X 0,Y 616.916,Z 184.321,A -85,B 0,C 180,E1 28918.735,E2 28918.735} C_VEL
LIN {X 0,Y 616.991,Z 184.316,A -85,B 0,C 180,E1 28915.703,E2 28915.703} C_VEL
LIN {X 0,Y 616.916,Z 184.32,A -85,B 0,C 180,E1 28912.687,E2 28912.687} C_VEL
LIN {X 0,Y 616.986,Z 184.315,A -85,B 0,C 180,E1 28909.682,E2 28909.682} C_VEL
LIN {X 0,Y 616.917,Z 184.32,A -85,B 0,C 180,E1 28906.687,E2 28906.687} C_VEL
LIN {X 0,Y 616.965,Z 184.319,A -85,B 0,C 180,E1 28903.589,E2 28903.589} C_VEL
LIN {X 0,Y 616.92,Z 184.322,A -85,B 0,C 180,E1 28900.646,E2 28900.646} C_VEL
LIN {X 0,Y 616.939,Z 184.32,A -85,B 0,C 180,E1 28897.449,E2 28897.449} C_VEL
LIN {X 0,Y 616.922,Z 184.32,A -85,B 0,C 180,E1 28894.648,E2 28894.648} C_VEL
LIN {X 0,Y 616.929,Z 184.322,A -85,B 0,C 180,E1 28891.393,E2 28891.393} C_VEL
LIN {X 0,Y 616.919,Z 184.322,A -85,B 0,C 180,E1 28888.793,E2 28888.793} C_VEL
LIN {X 0,Y 616.946,Z 184.319,A -85,B 0,C 180,E1 28885.632,E2 28885.632} C_VEL
LIN {X 0,Y 616.92,Z 184.322,A -85,B 0,C 180,E1 28882.832,E2 28882.832} C_VEL
LIN {X 0,Y 616.94,Z 184.321,A -85,B 0,C 180,E1 28879.637,E2 28879.637} C_VEL
LIN {X 0,Y 616.926,Z 184.319,A -85,B 0,C 180,E1 28876.791,E2 28876.791} C_VEL
LIN {X 0,Y 616.926,Z 184.32,A -85,B 0,C 180,E1 28873.525,E2 28873.525} C_VEL
LIN {X 0,Y 616.94,Z 184.321,A -85,B 0,C 180,E1 28870.696,E2 28870.696} C_VEL
LIN {X 0,Y 616.922,Z 184.32,A -85,B 0,C 180,E1 28867.515,E2 28867.515} C_VEL
LIN {X 0,Y 616.95,Z 184.318,A -85,B 0,C 180,E1 28864.672,E2 28864.672} C_VEL
LIN {X 0,Y 616.92,Z 184.321,A -85,B 0,C 180,E1 28861.547,E2 28861.547} C_VEL
LIN {X 0,Y 616.948,Z 184.318,A -85,B 0,C 180,E1 28858.765,E2 28858.765} C_VEL
LIN {X 0,Y 616.923,Z 184.32,A -85,B 0,C 180,E1 28855.671,E2 28855.671} C_VEL
LIN {X 0,Y 616.959,Z 184.319,A -85,B 0,C 180,E1 28852.727,E2 28852.727} C_VEL
LIN {X 0,Y 616.923,Z 184.318,A -85,B 0,C 180,E1 28849.714,E2 28849.714} C_VEL
LIN {X 0,Y 616.939,Z 184.319,A -85,B 0,C 180,E1 28846.966,E2 28846.966} C_VEL
LIN {X 0,Y 616.922,Z 184.319,A -85,B 0,C 180,E1 28843.794,E2 28843.794} C_VEL
LIN {X 0,Y 616.954,Z 184.318,A -85,B 0,C 180,E1 28840.902,E2 28840.902} C_VEL
LIN {X 0,Y 616.918,Z 184.317,A -85,B 0,C 180,E1 28837.782,E2 28837.782} C_VEL
LIN {X 0,Y 616.957,Z 184.286,A -85,B 0,C 180,E1 28834.897,E2 28834.897} C_VEL
LIN {X 0,Y 616.916,Z 184.319,A -85,B 0,C 180,E1 28831.787,E2 28831.787} C_VEL
LIN {X 0,Y 616.971,Z 184.285,A -85,B 0,C 180,E1 28828.878,E2 28828.878} C_VEL
LIN {X 0,Y 616.917,Z 184.308,A -85,B 0,C 180,E1 28825.848,E2 28825.848} C_VEL
LIN {X 0,Y 616.997,Z 184.311,A -85,B 0,C 180,E1 28822.783,E2 28822.783} C_VEL
LIN {X 0,Y 616.915,Z 184.317,A -85,B 0,C 180,E1 28819.8,E2 28819.8} C_VEL
LIN {X 0,Y 616.987,Z 184.305,A -85,B 0,C 180,E1 28816.736,E2 28816.736} C_VEL
LIN {X 0,Y 616.914,Z 184.315,A -85,B 0,C 180,E1 28813.784,E2 28813.784} C_VEL
LIN {X 0,Y 616.98,Z 184.314,A -85,B 0,C 180,E1 28810.741,E2 28810.741} C_VEL
LIN {X 0,Y 616.916,Z 184.31,A -85,B 0,C 180,E1 28807.825,E2 28807.825} C_VEL
LIN {X 0,Y 616.981,Z 184.317,A -85,B 0,C 180,E1 28804.834,E2 28804.834} C_VEL
LIN {X 0,Y 616.915,Z 184.306,A -85,B 0,C 180,E1 28801.858,E2 28801.858} C_VEL
LIN {X 0,Y 616.969,Z 184.312,A -85,B 0,C 180,E1 28798.793,E2 28798.793} C_VEL
LIN {X 0,Y 616.92,Z 184.311,A -85,B 0,C 180,E1 28795.817,E2 28795.817} C_VEL
LIN {X 0,Y 616.941,Z 184.304,A -85,B 0,C 180,E1 28792.633,E2 28792.633} C_VEL
LIN {X 0,Y 616.923,Z 184.316,A -85,B 0,C 180,E1 28789.824,E2 28789.824} C_VEL
LIN {X 0,Y 616.933,Z 184.313,A -85,B 0,C 180,E1 28786.599,E2 28786.599} C_VEL
LIN {X 0,Y 616.923,Z 184.317,A -85,B 0,C 180,E1 28783.91,E2 28783.91} C_VEL
LIN {X 0,Y 616.935,Z 184.318,A -85,B 0,C 180,E1 28780.693,E2 28780.693} C_VEL
LIN {X 0,Y 616.926,Z 184.31,A -85,B 0,C 180,E1 28777.913,E2 28777.913} C_VEL
LIN {X 0,Y 616.93,Z 184.312,A -85,B 0,C 180,E1 28774.667,E2 28774.667} C_VEL
LIN {X 0,Y 616.935,Z 184.283,A -85,B 0,C 180,E1 28771.831,E2 28771.831} C_VEL
LIN {X 0,Y 616.924,Z 184.318,A -85,B 0,C 180,E1 28768.65,E2 28768.65} C_VEL
LIN {X 0,Y 616.95,Z 184.304,A -85,B 0,C 180,E1 28765.779,E2 28765.779} C_VEL
LIN {X 0,Y 616.924,Z 184.319,A -85,B 0,C 180,E1 28762.687,E2 28762.687} C_VEL
LIN {X 0,Y 616.944,Z 184.301,A -85,B 0,C 180,E1 28759.896,E2 28759.896} C_VEL
LIN {X 0,Y 616.92,Z 184.313,A -85,B 0,C 180,E1 28756.718,E2 28756.718} C_VEL
LIN {X 0,Y 616.968,Z 184.318,A -85,B 0,C 180,E1 28753.782,E2 28753.782} C_VEL
LIN {X 0,Y 616.923,Z 184.323,A -85,B 0,C 180,E1 28750.774,E2 28750.774} C_VEL
LIN {X 0,Y 616.94,Z 184.267,A -85,B 0,C 180,E1 28748.009,E2 28748.009} C_VEL
LIN {X 0,Y 617.027,Z 184.563,A -85,B 0,C 180,E1 28745.636,E2 28745.636} C_VEL
LIN {X 0,Y 623.312,Z 205.147,A -85,B 0,C 180,E1 28743.228,E2 28743.228} C_VEL
LIN {X 0,Y 626.182,Z 215.751,A -85,B 0,C 180,E1 28742.064,E2 28742.064} C_VEL
LIN {X 0,Y 625.749,Z 223.787,A -85,B 0,C 180,E1 28741.335,E2 28741.335} C_VEL
LIN {X 0,Y 632.098,Z 253.588,A -85,B 0,C 180,E1 28740.578,E2 28740.578} C_VEL
LIN {X 0,Y 628.843,Z 520.485,A -85,B 0,C 180,E1 28737.33,E2 28737.33} C_VEL
LIN {X 0,Y 628.312,Z 539.812,A -85,B 0,C 180,E1 28737.012,E2 28737.012} C_VEL
LIN {X 0,Y 627.677,Z 557.378,A -85,B 0,C 180,E1 28736.613,E2 28736.613} C_VEL
LIN {X 0,Y 626.937,Z 574.574,A -85,B 0,C 180,E1 28736.112,E2 28736.112} C_VEL
LIN {X 0,Y 626.111,Z 590.754,A -85,B 0,C 180,E1 28735.538,E2 28735.538} C_VEL
LIN {X 0,Y 625.215,Z 606.62,A -85,B 0,C 180,E1 28734.869,E2 28734.869} C_VEL
LIN {X 0,Y 624.204,Z 622.916,A -85,B 0,C 180,E1 28734.067,E2 28734.067} C_VEL
LIN {X 0,Y 622.96,Z 642.263,A -85,B 0,C 180,E1 28732.953,E2 28732.953} C_VEL
LIN {X 0,Y 621.686,Z 660.26,A -85,B 0,C 180,E1 28731.708,E2 28731.708} C_VEL
LIN {X 0,Y 620.663,Z 674.743,A -85,B 0,C 180,E1 28730.558,E2 28730.558} C_VEL
LIN {X 0,Y 619.753,Z 688.042,A -85,B 0,C 180,E1 28729.36,E2 28729.36} C_VEL
LIN {X 0,Y 618.901,Z 700.723,A -85,B 0,C 180,E1 28728.068,E2 28728.068} C_VEL
LIN {X 0,Y 618.135,Z 713.111,A -85,B 0,C 180,E1 28726.635,E2 28726.635} C_VEL
LIN {X 0,Y 617.344,Z 727.236,A -85,B 0,C 180,E1 28724.729,E2 28724.729} C_VEL
LIN {X 0,Y 616.828,Z 737.343,A -85,B 0,C 180,E1 28723.115,E2 28723.115} C_VEL
LIN {X 0,Y 616.487,Z 745.634,A -85,B 0,C 180,E1 28721.58,E2 28721.58} C_VEL
LIN {X 0,Y 616.257,Z 752.537,A -85,B 0,C 180,E1 28720.091,E2 28720.091} C_VEL
LIN {X 0,Y 616.087,Z 758.436,A -85,B 0,C 180,E1 28718.586,E2 28718.586} C_VEL
LIN {X 0,Y 615.984,Z 763.568,A -85,B 0,C 180,E1 28716.992,E2 28716.992} C_VEL
LIN {X 0,Y 615.944,Z 767.356,A -85,B 0,C 180,E1 28715.495,E2 28715.495} C_VEL
LIN {X 0,Y 615.923,Z 770.349,A -85,B 0,C 180,E1 28713.909,E2 28713.909} C_VEL
LIN {X 0,Y 615.91,Z 772.317,A -85,B 0,C 180,E1 28712.326,E2 28712.326} C_VEL
LIN {X 0,Y 615.908,Z 773.281,A -85,B 0,C 180,E1 28710.744,E2 28710.744} C_VEL
LIN {X 0,Y 615.91,Z 773.252,A -85,B 0,C 180,E1 28709.163,E2 28709.163} C_VEL
LIN {X 0,Y 615.912,Z 772.143,A -85,B 0,C 180,E1 28707.488,E2 28707.488} C_VEL
LIN {X 0,Y 615.926,Z 769.765,A -85,B 0,C 180,E1 28705.718,E2 28705.718} C_VEL
LIN {X 0,Y 615.972,Z 764.909,A -85,B 0,C 180,E1 28703.476,E2 28703.476} C_VEL
LIN {X 0,Y 616.079,Z 759.435,A -85,B 0,C 180,E1 28701.696,E2 28701.696} C_VEL
LIN {X 0,Y 616.228,Z 753.335,A -85,B 0,C 180,E1 28700.098,E2 28700.098} C_VEL
LIN {X 0,Y 616.451,Z 746.47,A -85,B 0,C 180,E1 28698.588,E2 28698.588} C_VEL
LIN {X 0,Y 616.783,Z 738.425,A -85,B 0,C 180,E1 28697.074,E2 28697.074} C_VEL
LIN {X 0,Y 617.202,Z 729.688,A -85,B 0,C 180,E1 28695.647,E2 28695.647} C_VEL
LIN {X 0,Y 617.741,Z 719.739,A -85,B 0,C 180,E1 28694.223,E2 28694.223} C_VEL
LIN {X 0,Y 618.479,Z 707.569,A -85,B 0,C 180,E1 28692.697,E2 28692.697} C_VEL
LIN {X 0,Y 619.552,Z 691.041,A -85,B 0,C 180,E1 28690.927,E2 28690.927} C_VEL
LIN {X 0,Y 620.519,Z 676.987,A -85,B 0,C 180,E1 28689.634,E2 28689.634} C_VEL
LIN {X 0,Y 621.437,Z 663.628,A -85,B 0,C 180,E1 28688.548,E2 28688.548} C_VEL
LIN {X 0,Y 622.428,Z 649.398,A -85,B 0,C 180,E1 28687.525,E2 28687.525} C_VEL
LIN {X 0,Y 623.413,Z 635.02,A -85,B 0,C 180,E1 28686.615,E2 28686.615} C_VEL
LIN {X 0,Y 624.362,Z 620.37,A -85,B 0,C 180,E1 28685.8,E2 28685.8} C_VEL
LIN {X 0,Y 625.326,Z 604.697,A -85,B 0,C 180,E1 28685.044,E2 28685.044} C_VEL
LIN {X 0,Y 626.24,Z 588.229,A -85,B 0,C 180,E1 28684.365,E2 28684.365} C_VEL
LIN {X 0,Y 627.188,Z 569.368,A -85,B 0,C 180,E1 28683.721,E2 28683.721} C_VEL
LIN {X 0,Y 628.15,Z 545.459,A -85,B 0,C 180,E1 28683.103,E2 28683.103} C_VEL
LIN {X 0,Y 628.703,Z 526.452,A -85,B 0,C 180,E1 28682.757,E2 28682.757} C_VEL
LIN {X 0,Y 629.775,Z 444.459,A -85,B 0,C 180,E1 28681.744,E2 28681.744} C_VEL
LIN {X 0,Y 631.974,Z 252.058,A -85,B 0,C 180,E1 28679.396,E2 28679.396} C_VEL
LIN {X 0,Y 625.75,Z 223.79,A -85,B 0,C 180,E1 28678.665,E2 28678.665} C_VEL
LIN {X 0,Y 626.077,Z 214.688,A -85,B 0,C 180,E1 28677.828,E2 28677.828} C_VEL
LIN {X 0,Y 619.621,Z 193.091,A -85,B 0,C 180,E1 28675.386,E2 28675.386} C_VEL
LIN {X 0,Y 617.007,Z 184.442,A -85,B 0,C 180,E1 28674.331,E2 28674.331} C_VEL
LIN {X 0,Y 616.911,Z 184.282,A -85,B 0,C 180,E1 28671.373,E2 28671.373} C_VEL
LIN {X 0,Y 616.986,Z 184.303,A -85,B 0,C 180,E1 28668.34,E2 28668.34} C_VEL
LIN {X 0,Y 616.918,Z 184.318,A -85,B 0,C 180,E1 28665.359,E2 28665.359} C_VEL
LIN {X 0,Y 616.967,Z 184.318,A -85,B 0,C 180,E1 28662.266,E2 28662.266} C_VEL
LIN {X 0,Y 616.916,Z 184.306,A -85,B 0,C 180,E1 28659.446,E2 28659.446} C_VEL
LIN {X 0,Y 616.974,Z 184.306,A -85,B 0,C 180,E1 28656.381,E2 28656.381} C_VEL
LIN {X 0,Y 616.919,Z 184.311,A -85,B 0,C 180,E1 28653.427,E2 28653.427} C_VEL
LIN {X 0,Y 616.949,Z 184.302,A -85,B 0,C 180,E1 28650.264,E2 28650.264} C_VEL
LIN {X 0,Y 616.921,Z 184.289,A -85,B 0,C 180,E1 28647.407,E2 28647.407} C_VEL
LIN {X 0,Y 616.936,Z 184.317,A -85,B 0,C 180,E1 28644.168,E2 28644.168} C_VEL
LIN {X 0,Y 616.927,Z 184.309,A -85,B 0,C 180,E1 28641.387,E2 28641.387} C_VEL
LIN {X 0,Y 616.927,Z 184.306,A -85,B 0,C 180,E1 28638.131,E2 28638.131} C_VEL
LIN {X 0,Y 616.938,Z 184.315,A -85,B 0,C 180,E1 28635.318,E2 28635.318} C_VEL
LIN {X 0,Y 616.924,Z 184.312,A -85,B 0,C 180,E1 28632.163,E2 28632.163} C_VEL
LIN {X 0,Y 616.95,Z 184.315,A -85,B 0,C 180,E1 28629.295,E2 28629.295} C_VEL
LIN {X 0,Y 616.92,Z 184.317,A -85,B 0,C 180,E1 28626.141,E2 28626.141} C_VEL
LIN {X 0,Y 616.96,Z 184.309,A -85,B 0,C 180,E1 28623.252,E2 28623.252} C_VEL
LIN {X 0,Y 616.918,Z 184.317,A -85,B 0,C 180,E1 28620.186,E2 28620.186} C_VEL
LIN {X 0,Y 616.96,Z 184.305,A -85,B 0,C 180,E1 28617.306,E2 28617.306} C_VEL
LIN {X 0,Y 616.916,Z 184.315,A -85,B 0,C 180,E1 28614.233,E2 28614.233} C_VEL
LIN {X 0,Y 616.955,Z 184.311,A -85,B 0,C 180,E1 28611.425,E2 28611.425} C_VEL
LIN {X 0,Y 616.917,Z 184.308,A -85,B 0,C 180,E1 28608.311,E2 28608.311} C_VEL
LIN {X 0,Y 616.971,Z 184.317,A -85,B 0,C 180,E1 28605.356,E2 28605.356} C_VEL
LIN {X 0,Y 616.918,Z 184.313,A -85,B 0,C 180,E1 28602.343,E2 28602.343} C_VEL
LIN {X 0,Y 616.976,Z 184.313,A -85,B 0,C 180,E1 28599.41,E2 28599.41} C_VEL
LIN {X 0,Y 616.917,Z 184.318,A -85,B 0,C 180,E1 28596.401,E2 28596.401} C_VEL
LIN {X 0,Y 616.978,Z 184.286,A -85,B 0,C 180,E1 28593.43,E2 28593.43} C_VEL
LIN {X 0,Y 616.915,Z 184.308,A -85,B 0,C 180,E1 28590.374,E2 28590.374} C_VEL
LIN {X 0,Y 616.989,Z 184.311,A -85,B 0,C 180,E1 28587.415,E2 28587.415} C_VEL
LIN {X 0,Y 616.91,Z 184.293,A -85,B 0,C 180,E1 28584.418,E2 28584.418} C_VEL
LIN {X 0,Y 616.994,Z 184.316,A -85,B 0,C 180,E1 28581.353,E2 28581.353} C_VEL
LIN {X 0,Y 616.916,Z 184.318,A -85,B 0,C 180,E1 28578.478,E2 28578.478} C_VEL
LIN {X 0,Y 616.988,Z 184.318,A -85,B 0,C 180,E1 28575.435,E2 28575.435} C_VEL
LIN {X 0,Y 616.918,Z 184.319,A -85,B 0,C 180,E1 28572.388,E2 28572.388} C_VEL
LIN {X 0,Y 616.967,Z 184.318,A -85,B 0,C 180,E1 28569.315,E2 28569.315} C_VEL
LIN {X 0,Y 616.917,Z 184.318,A -85,B 0,C 180,E1 28566.495,E2 28566.495} C_VEL
LIN {X 0,Y 616.917,Z 184.32,A -85,B 0,C 180,E1 28564.763,E2 28564.763} C_VEL
LIN {X 0,Y 615.944,Z 184.445,A -85,B 0,C 180,E1 28564.048,E2 28564.048} C_VEL
LIN {X 0,Y 609.523,Z 185.252,A -85,B 0,C 180,E1 28561.989,E2 28561.989} C_VEL
LIN {X 0,Y 609.042,Z 185.306,A -85,B 0,C 180,E1 28561.519,E2 28561.519} C_VEL
LIN {X 0,Y 608.98,Z 185.31,A -85,B 0,C 180,E1 28558.537,E2 28558.537} C_VEL
LIN {X 0,Y 609.024,Z 185.306,A -85,B 0,C 180,E1 28555.446,E2 28555.446} C_VEL
LIN {X 0,Y 608.98,Z 185.31,A -85,B 0,C 180,E1 28552.591,E2 28552.591} C_VEL
LIN {X 0,Y 609.019,Z 185.308,A -85,B 0,C 180,E1 28549.466,E2 28549.466} C_VEL
LIN {X 0,Y 608.981,Z 185.309,A -85,B 0,C 180,E1 28546.598,E2 28546.598} C_VEL
LIN {X 0,Y 609.012,Z 185.308,A -85,B 0,C 180,E1 28543.48,E2 28543.48} C_VEL
LIN {X 0,Y 608.984,Z 185.312,A -85,B 0,C 180,E1 28540.595,E2 28540.595} C_VEL
LIN {X 0,Y 608.994,Z 185.309,A -85,B 0,C 180,E1 28537.357,E2 28537.357} C_VEL
LIN {X 0,Y 608.993,Z 185.308,A -85,B 0,C 180,E1 28534.52,E2 28534.52} C_VEL
LIN {X 0,Y 608.985,Z 185.311,A -85,B 0,C 180,E1 28531.317,E2 28531.317} C_VEL
LIN {X 0,Y 608.985,Z 185.311,A -85,B 0,C 180,E1 28528.683,E2 28528.683} C_VEL
LIN {X 0,Y 608.985,Z 185.309,A -85,B 0,C 180,E1 28525.386,E2 28525.386} C_VEL
LIN {X 0,Y 609.001,Z 185.308,A -85,B 0,C 180,E1 28522.548,E2 28522.548} C_VEL
LIN {X 0,Y 608.984,Z 185.312,A -85,B 0,C 180,E1 28519.405,E2 28519.405} C_VEL
LIN {X 0,Y 609.012,Z 185.308,A -85,B 0,C 180,E1 28516.52,E2 28516.52} C_VEL
LIN {X 0,Y 608.981,Z 185.309,A -85,B 0,C 180,E1 28513.402,E2 28513.402} C_VEL
LIN {X 0,Y 609.032,Z 185.306,A -85,B 0,C 180,E1 28510.435,E2 28510.435} C_VEL
LIN {X 0,Y 608.98,Z 185.31,A -85,B 0,C 180,E1 28507.409,E2 28507.409} C_VEL
LIN {X 0,Y 609.041,Z 185.305,A -85,B 0,C 180,E1 28504.423,E2 28504.423} C_VEL
LIN {X 0,Y 608.978,Z 185.31,A -85,B 0,C 180,E1 28501.356,E2 28501.356} C_VEL
LIN {X 0,Y 609.053,Z 185.305,A -85,B 0,C 180,E1 28498.313,E2 28498.313} C_VEL
LIN {X 0,Y 608.977,Z 185.309,A -85,B 0,C 180,E1 28495.273,E2 28495.273} C_VEL
LIN {X 0,Y 609.019,Z 185.307,A -85,B 0,C 180,E1 28492.124,E2 28492.124} C_VEL
LIN {X 0,Y 608.979,Z 185.308,A -85,B 0,C 180,E1 28489.326,E2 28489.326} C_VEL
LIN {X 0,Y 609.028,Z 185.307,A -85,B 0,C 180,E1 28486.252,E2 28486.252} C_VEL
LIN {X 0,Y 608.98,Z 185.308,A -85,B 0,C 180,E1 28483.34,E2 28483.34} C_VEL
LIN {X 0,Y 609.011,Z 185.308,A -85,B 0,C 180,E1 28480.184,E2 28480.184} C_VEL
LIN {X 0,Y 608.98,Z 185.306,A -85,B 0,C 180,E1 28477.385,E2 28477.385} C_VEL
LIN {X 0,Y 609,Z 185.285,A -85,B 0,C 180,E1 28474.161,E2 28474.161} C_VEL
LIN {X 0,Y 608.985,Z 185.308,A -85,B 0,C 180,E1 28471.365,E2 28471.365} C_VEL
LIN {X 0,Y 608.989,Z 185.263,A -85,B 0,C 180,E1 28468.114,E2 28468.114} C_VEL
LIN {X 0,Y 608.998,Z 185.296,A -85,B 0,C 180,E1 28465.239,E2 28465.239} C_VEL
LIN {X 0,Y 608.986,Z 185.298,A -85,B 0,C 180,E1 28462.086,E2 28462.086} C_VEL
LIN {X 0,Y 609.002,Z 185.306,A -85,B 0,C 180,E1 28459.27,E2 28459.27} C_VEL
LIN {X 0,Y 608.983,Z 185.302,A -85,B 0,C 180,E1 28456.11,E2 28456.11} C_VEL
LIN {X 0,Y 608.996,Z 185.304,A -85,B 0,C 180,E1 28453.386,E2 28453.386} C_VEL
LIN {X 0,Y 608.986,Z 185.306,A -85,B 0,C 180,E1 28450.214,E2 28450.214} C_VEL
LIN {X 0,Y 609.006,Z 185.297,A -85,B 0,C 180,E1 28447.358,E2 28447.358} C_VEL
LIN {X 0,Y 608.982,Z 185.305,A -85,B 0,C 180,E1 28444.237,E2 28444.237} C_VEL
LIN {X 0,Y 609.016,Z 185.294,A -85,B 0,C 180,E1 28441.317,E2 28441.317} C_VEL
LIN {X 0,Y 608.979,Z 185.3,A -85,B 0,C 180,E1 28438.212,E2 28438.212} C_VEL
LIN {X 0,Y 609.041,Z 185.301,A -85,B 0,C 180,E1 28435.197,E2 28435.197} C_VEL
LIN {X 0,Y 608.977,Z 185.292,A -85,B 0,C 180,E1 28432.167,E2 28432.167} C_VEL
LIN {X 0,Y 609.051,Z 185.302,A -85,B 0,C 180,E1 28429.117,E2 28429.117} C_VEL
LIN {X 0,Y 608.977,Z 185.302,A -85,B 0,C 180,E1 28426.13,E2 28426.13} C_VEL
LIN {X 0,Y 609.048,Z 185.294,A -85,B 0,C 180,E1 28423.107,E2 28423.107} C_VEL
LIN {X 0,Y 608.978,Z 185.307,A -85,B 0,C 180,E1 28420.131,E2 28420.131} C_VEL
LIN {X 0,Y 609.035,Z 185.301,A -85,B 0,C 180,E1 28417.058,E2 28417.058} C_VEL
LIN {X 0,Y 608.981,Z 185.301,A -85,B 0,C 180,E1 28414.103,E2 28414.103} C_VEL
LIN {X 0,Y 609.006,Z 185.276,A -85,B 0,C 180,E1 28410.923,E2 28410.923} C_VEL
LIN {X 0,Y 608.986,Z 185.307,A -85,B 0,C 180,E1 28408.075,E2 28408.075} C_VEL
LIN {X 0,Y 608.99,Z 185.289,A -85,B 0,C 180,E1 28404.809,E2 28404.809} C_VEL
LIN {X 0,Y 608.996,Z 185.308,A -85,B 0,C 180,E1 28401.997,E2 28401.997} C_VEL
LIN {X 0,Y 608.986,Z 185.306,A -85,B 0,C 180,E1 28398.754,E2 28398.754} C_VEL
LIN {X 0,Y 609.017,Z 185.292,A -85,B 0,C 180,E1 28395.838,E2 28395.838} C_VEL
LIN {X 0,Y 608.98,Z 185.301,A -85,B 0,C 180,E1 28392.689,E2 28392.689} C_VEL
LIN {X 0,Y 609.031,Z 185.296,A -85,B 0,C 180,E1 28389.794,E2 28389.794} C_VEL
LIN {X 0,Y 608.974,Z 185.261,A -85,B 0,C 180,E1 28386.697,E2 28386.697} C_VEL
LIN {X 0,Y 609.061,Z 185.653,A -85,B 0,C 180,E1 28386.034,E2 28386.034} C_VEL
LIN {X 0,Y 615.515,Z 206.449,A -85,B 0,C 180,E1 28383.554,E2 28383.554} C_VEL
LIN {X 0,Y 618.759,Z 218.365,A -85,B 0,C 180,E1 28382.221,E2 28382.221} C_VEL
LIN {X 0,Y 618.47,Z 223.597,A -85,B 0,C 180,E1 28381.745,E2 28381.745} C_VEL
LIN {X 0,Y 625.184,Z 254.844,A -85,B 0,C 180,E1 28380.934,E2 28380.934} C_VEL
LIN {X 0,Y 621.721,Z 520.72,A -85,B 0,C 180,E1 28377.663,E2 28377.663} C_VEL
LIN {X 0,Y 621.171,Z 539.637,A -85,B 0,C 180,E1 28377.348,E2 28377.348} C_VEL
LIN {X 0,Y 620.495,Z 557.167,A -85,B 0,C 180,E1 28376.946,E2 28376.946} C_VEL
LIN {X 0,Y 619.704,Z 574.398,A -85,B 0,C 180,E1 28376.44,E2 28376.44} C_VEL
LIN {X 0,Y 618.793,Z 591.205,A -85,B 0,C 180,E1 28375.836,E2 28375.836} C_VEL
LIN {X 0,Y 617.745,Z 608.569,A -85,B 0,C 180,E1 28375.089,E2 28375.089} C_VEL
LIN {X 0,Y 616.376,Z 629.197,A -85,B 0,C 180,E1 28374.024,E2 28374.024} C_VEL
LIN {X 0,Y 615.078,Z 647.086,A -85,B 0,C 180,E1 28372.91,E2 28372.91} C_VEL
LIN {X 0,Y 614.014,Z 661.343,A -85,B 0,C 180,E1 28371.892,E2 28371.892} C_VEL
LIN {X 0,Y 612.975,Z 675.125,A -85,B 0,C 180,E1 28370.777,E2 28370.777} C_VEL
LIN {X 0,Y 612.043,Z 687.864,A -85,B 0,C 180,E1 28369.614,E2 28369.614} C_VEL
LIN {X 0,Y 611.134,Z 700.544,A -85,B 0,C 180,E1 28368.306,E2 28368.306} C_VEL
LIN {X 0,Y 610.306,Z 712.933,A -85,B 0,C 180,E1 28366.855,E2 28366.855} C_VEL
LIN {X 0,Y 609.445,Z 727.182,A -85,B 0,C 180,E1 28364.905,E2 28364.905} C_VEL
LIN {X 0,Y 608.899,Z 737.165,A -85,B 0,C 180,E1 28363.289,E2 28363.289} C_VEL
LIN {X 0,Y 608.537,Z 745.357,A -85,B 0,C 180,E1 28361.754,E2 28361.754} C_VEL
LIN {X 0,Y 608.284,Z 752.36,A -85,B 0,C 180,E1 28360.224,E2 28360.224} C_VEL
LIN {X 0,Y 608.098,Z 758.259,A -85,B 0,C 180,E1 28358.7,E2 28358.7} C_VEL
LIN {X 0,Y 607.993,Z 763.392,A -85,B 0,C 180,E1 28357.084,E2 28357.084} C_VEL
LIN {X 0,Y 607.946,Z 767.21,A -85,B 0,C 180,E1 28355.568,E2 28355.568} C_VEL
LIN {X 0,Y 607.924,Z 770.232,A -85,B 0,C 180,E1 28353.961,E2 28353.961} C_VEL
LIN {X 0,Y 607.911,Z 772.22,A -85,B 0,C 180,E1 28352.356,E2 28352.356} C_VEL
LIN {X 0,Y 607.908,Z 773.194,A -85,B 0,C 180,E1 28350.754,E2 28350.754} C_VEL
LIN {X 0,Y 607.91,Z 773.165,A -85,B 0,C 180,E1 28349.152,E2 28349.152} C_VEL
LIN {X 0,Y 607.911,Z 772.132,A -85,B 0,C 180,E1 28347.549,E2 28347.549} C_VEL
LIN {X 0,Y 607.925,Z 770.085,A -85,B 0,C 180,E1 28345.945,E2 28345.945} C_VEL
LIN {X 0,Y 607.951,Z 766.795,A -85,B 0,C 180,E1 28344.243,E2 28344.243} C_VEL
LIN {X 0,Y 608.026,Z 761.776,A -85,B 0,C 180,E1 28342.346,E2 28342.346} C_VEL
LIN {X 0,Y 608.212,Z 754.355,A -85,B 0,C 180,E1 28340.252,E2 28340.252} C_VEL
LIN {X 0,Y 608.474,Z 746.761,A -85,B 0,C 180,E1 28338.533,E2 28338.533} C_VEL
LIN {X 0,Y 608.822,Z 738.788,A -85,B 0,C 180,E1 28336.999,E2 28336.999} C_VEL
LIN {X 0,Y 609.278,Z 729.947,A -85,B 0,C 180,E1 28335.525,E2 28335.525} C_VEL
LIN {X 0,Y 609.839,Z 720.262,A -85,B 0,C 180,E1 28334.111,E2 28334.111} C_VEL
LIN {X 0,Y 610.534,Z 709.354,A -85,B 0,C 180,E1 28332.708,E2 28332.708} C_VEL
LIN {X 0,Y 611.442,Z 696.317,A -85,B 0,C 180,E1 28331.234,E2 28331.234} C_VEL
LIN {X 0,Y 612.707,Z 679.053,A -85,B 0,C 180,E1 28329.563,E2 28329.563} C_VEL
LIN {X 0,Y 613.772,Z 664.497,A -85,B 0,C 180,E1 28328.35,E2 28328.35} C_VEL
LIN {X 0,Y 614.857,Z 649.931,A -85,B 0,C 180,E1 28327.283,E2 28327.283} C_VEL
LIN {X 0,Y 615.901,Z 635.649,A -85,B 0,C 180,E1 28326.363,E2 28326.363} C_VEL
LIN {X 0,Y 616.967,Z 620.193,A -85,B 0,C 180,E1 28325.491,E2 28325.491} C_VEL
LIN {X 0,Y 617.954,Z 605.166,A -85,B 0,C 180,E1 28324.757,E2 28324.757} C_VEL
LIN {X 0,Y 618.895,Z 589.298,A -85,B 0,C 180,E1 28324.09,E2 28324.09} C_VEL
LIN {X 0,Y 619.776,Z 572.91,A -85,B 0,C 180,E1 28323.511,E2 28323.511} C_VEL
LIN {X 0,Y 620.582,Z 555.243,A -85,B 0,C 180,E1 28323.003,E2 28323.003} C_VEL
LIN {X 0,Y 621.431,Z 533.591,A -85,B 0,C 180,E1 28322.531,E2 28322.531} C_VEL
LIN {X 0,Y 622.005,Z 501.727,A -85,B 0,C 180,E1 28322.095,E2 28322.095} C_VEL
LIN {X 0,Y 625.137,Z 253.881,A -85,B 0,C 180,E1 28319.051,E2 28319.051} C_VEL
LIN {X 0,Y 618.469,Z 223.599,A -85,B 0,C 180,E1 28318.255,E2 28318.255} C_VEL
LIN {X 0,Y 618.643,Z 217.229,A -85,B 0,C 180,E1 28317.662,E2 28317.662} C_VEL
LIN {X 0,Y 612.32,Z 196.001,A -85,B 0,C 180,E1 28315.223,E2 28315.223} C_VEL
LIN {X 0,Y 609.023,Z 185.441,A -85,B 0,C 180,E1 28313.92,E2 28313.92} C_VEL
LIN {X 0,Y 608.98,Z 185.273,A -85,B 0,C 180,E1 28311.162,E2 28311.162} C_VEL
LIN {X 0,Y 608.998,Z 185.295,A -85,B 0,C 180,E1 28307.949,E2 28307.949} C_VEL
LIN {X 0,Y 608.996,Z 185.301,A -85,B 0,C 180,E1 28305.044,E2 28305.044} C_VEL
LIN {X 0,Y 608.986,Z 185.306,A -85,B 0,C 180,E1 28301.806,E2 28301.806} C_VEL
LIN {X 0,Y 608.999,Z 185.295,A -85,B 0,C 180,E1 28299.059,E2 28299.059} C_VEL
LIN {X 0,Y 608.985,Z 185.294,A -85,B 0,C 180,E1 28295.885,E2 28295.885} C_VEL
LIN {X 0,Y 609.014,Z 185.3,A -85,B 0,C 180,E1 28292.981,E2 28292.981} C_VEL
LIN {X 0,Y 608.98,Z 185.291,A -85,B 0,C 180,E1 28289.91,E2 28289.91} C_VEL
LIN {X 0,Y 609.013,Z 185.276,A -85,B 0,C 180,E1 28287.051,E2 28287.051} C_VEL
LIN {X 0,Y 608.981,Z 185.306,A -85,B 0,C 180,E1 28283.926,E2 28283.926} C_VEL
LIN {X 0,Y 609.02,Z 185.297,A -85,B 0,C 180,E1 28281.073,E2 28281.073} C_VEL
LIN {X 0,Y 608.98,Z 185.295,A -85,B 0,C 180,E1 28277.98,E2 28277.98} C_VEL
LIN {X 0,Y 609.048,Z 185.304,A -85,B 0,C 180,E1 28274.937,E2 28274.937} C_VEL
LIN {X 0,Y 608.977,Z 185.301,A -85,B 0,C 180,E1 28271.844,E2 28271.844} C_VEL
LIN {X 0,Y 609.045,Z 185.292,A -85,B 0,C 180,E1 28268.782,E2 28268.782} C_VEL
LIN {X 0,Y 608.978,Z 185.306,A -85,B 0,C 180,E1 28265.81,E2 28265.81} C_VEL
LIN {X 0,Y 609.027,Z 185.296,A -85,B 0,C 180,E1 28262.729,E2 28262.729} C_VEL
LIN {X 0,Y 608.979,Z 185.306,A -85,B 0,C 180,E1 28259.812,E2 28259.812} C_VEL
LIN {X 0,Y 609.017,Z 185.305,A -85,B 0,C 180,E1 28256.706,E2 28256.706} C_VEL
LIN {X 0,Y 608.982,Z 185.303,A -85,B 0,C 180,E1 28253.779,E2 28253.779} C_VEL
LIN {X 0,Y 608.995,Z 185.307,A -85,B 0,C 180,E1 28250.55,E2 28250.55} C_VEL
LIN {X 0,Y 608.994,Z 185.296,A -85,B 0,C 180,E1 28247.676,E2 28247.676} C_VEL
LIN {X 0,Y 608.983,Z 185.303,A -85,B 0,C 180,E1 28244.477,E2 28244.477} C_VEL
LIN {X 0,Y 609.009,Z 185.302,A -85,B 0,C 180,E1 28241.595,E2 28241.595} C_VEL
LIN {X 0,Y 608.983,Z 185.298,A -85,B 0,C 180,E1 28238.522,E2 28238.522} C_VEL
LIN {X 0,Y 609.012,Z 185.307,A -85,B 0,C 180,E1 28235.656,E2 28235.656} C_VEL
LIN {X 0,Y 608.976,Z 185.266,A -85,B 0,C 180,E1 28232.524,E2 28232.524} C_VEL
LIN {X 0,Y 609.022,Z 185.297,A -85,B 0,C 180,E1 28229.624,E2 28229.624} C_VEL
LIN {X 0,Y 608.978,Z 185.296,A -85,B 0,C 180,E1 28226.51,E2 28226.51} C_VEL
LIN {X 0,Y 609.038,Z 185.282,A -85,B 0,C 180,E1 28223.536,E2 28223.536} C_VEL
LIN {X 0,Y 608.978,Z 185.308,A -85,B 0,C 180,E1 28220.497,E2 28220.497} C_VEL
LIN {X 0,Y 609.053,Z 185.305,A -85,B 0,C 180,E1 28217.479,E2 28217.479} C_VEL
LIN {X 0,Y 608.977,Z 185.309,A -85,B 0,C 180,E1 28214.419,E2 28214.419} C_VEL
LIN {X 0,Y 609.028,Z 185.306,A -85,B 0,C 180,E1 28211.293,E2 28211.293} C_VEL
LIN {X 0,Y 608.978,Z 185.309,A -85,B 0,C 180,E1 28208.446,E2 28208.446} C_VEL
LIN {X 0,Y 609.024,Z 185.306,A -85,B 0,C 180,E1 28205.316,E2 28205.316} C_VEL
LIN {X 0,Y 608.984,Z 185.309,A -85,B 0,C 180,E1 28202.356,E2 28202.356} C_VEL
LIN {X 0,Y 609.042,Z 185.306,A -85,B 0,C 180,E1 28201.519,E2 28201.519} C_VEL
LIN {X 0,Y 607.974,Z 185.435,A -85,B 0,C 180,E1 28200.794,E2 28200.794} C_VEL
LIN {X 0,Y 601.547,Z 186.237,A -85,B 0,C 180,E1 28198.762,E2 28198.762} C_VEL
LIN {X 0,Y 601.056,Z 186.299,A -85,B 0,C 180,E1 28198.233,E2 28198.233} C_VEL
LIN {X 0,Y 601.046,Z 186.299,A -85,B 0,C 180,E1 28194.992,E2 28194.992} C_VEL
LIN {X 0,Y 601.078,Z 186.296,A -85,B 0,C 180,E1 28192.08,E2 28192.08} C_VEL
LIN {X 0,Y 601.04,Z 186.3,A -85,B 0,C 180,E1 28188.927,E2 28188.927} C_VEL
LIN {X 0,Y 601.115,Z 186.292,A -85,B 0,C 180,E1 28185.829,E2 28185.829} C_VEL
LIN {X 0,Y 601.037,Z 186.298,A -85,B 0,C 180,E1 28182.781,E2 28182.781} C_VEL
LIN {X 0,Y 601.09,Z 186.297,A -85,B 0,C 180,E1 28179.671,E2 28179.671} C_VEL
LIN {X 0,Y 601.039,Z 186.301,A -85,B 0,C 180,E1 28176.782,E2 28176.782} C_VEL
LIN {X 0,Y 601.074,Z 186.296,A -85,B 0,C 180,E1 28173.624,E2 28173.624} C_VEL
LIN {X 0,Y 601.047,Z 186.298,A -85,B 0,C 180,E1 28170.667,E2 28170.667} C_VEL
LIN {X 0,Y 601.046,Z 186.301,A -85,B 0,C 180,E1 28167.331,E2 28167.331} C_VEL
LIN {X 0,Y 601.08,Z 186.298,A -85,B 0,C 180,E1 28164.368,E2 28164.368} C_VEL
LIN {X 0,Y 601.04,Z 186.298,A -85,B 0,C 180,E1 28161.294,E2 28161.294} C_VEL
LIN {X 0,Y 601.097,Z 186.294,A -85,B 0,C 180,E1 28158.293,E2 28158.293} C_VEL
LIN {X 0,Y 601.038,Z 186.301,A -85,B 0,C 180,E1 28155.256,E2 28155.256} C_VEL
LIN {X 0,Y 601.112,Z 186.294,A -85,B 0,C 180,E1 28152.18,E2 28152.18} C_VEL
LIN {X 0,Y 601.039,Z 186.299,A -85,B 0,C 180,E1 28149.148,E2 28149.148} C_VEL
LIN {X 0,Y 601.094,Z 186.294,A -85,B 0,C 180,E1 28146.057,E2 28146.057} C_VEL
LIN {X 0,Y 601.044,Z 186.297,A -85,B 0,C 180,E1 28143.086,E2 28143.086} C_VEL
LIN {X 0,Y 601.064,Z 186.297,A -85,B 0,C 180,E1 28139.887,E2 28139.887} C_VEL
LIN {X 0,Y 601.053,Z 186.298,A -85,B 0,C 180,E1 28136.976,E2 28136.976} C_VEL
LIN {X 0,Y 601.046,Z 186.297,A -85,B 0,C 180,E1 28133.69,E2 28133.69} C_VEL
LIN {X 0,Y 601.074,Z 186.297,A -85,B 0,C 180,E1 28130.799,E2 28130.799} C_VEL
LIN {X 0,Y 601.042,Z 186.297,A -85,B 0,C 180,E1 28127.65,E2 28127.65} C_VEL
LIN {X 0,Y 601.109,Z 186.296,A -85,B 0,C 180,E1 28124.585,E2 28124.585} C_VEL
LIN {X 0,Y 601.039,Z 186.297,A -85,B 0,C 180,E1 28121.538,E2 28121.538} C_VEL
LIN {X 0,Y 601.12,Z 186.294,A -85,B 0,C 180,E1 28118.585,E2 28118.585} C_VEL
LIN {X 0,Y 601.034,Z 186.266,A -85,B 0,C 180,E1 28115.493,E2 28115.493} C_VEL
LIN {X 0,Y 601.081,Z 186.297,A -85,B 0,C 180,E1 28112.335,E2 28112.335} C_VEL
LIN {X 0,Y 601.039,Z 186.286,A -85,B 0,C 180,E1 28109.5,E2 28109.5} C_VEL
LIN {X 0,Y 601.075,Z 186.268,A -85,B 0,C 180,E1 28106.369,E2 28106.369} C_VEL
LIN {X 0,Y 601.048,Z 186.296,A -85,B 0,C 180,E1 28103.428,E2 28103.428} C_VEL
LIN {X 0,Y 601.051,Z 186.295,A -85,B 0,C 180,E1 28100.143,E2 28100.143} C_VEL
LIN {X 0,Y 601.069,Z 186.287,A -85,B 0,C 180,E1 28097.224,E2 28097.224} C_VEL
LIN {X 0,Y 601.04,Z 186.293,A -85,B 0,C 180,E1 28094.057,E2 28094.057} C_VEL
LIN {X 0,Y 601.099,Z 186.285,A -85,B 0,C 180,E1 28091.028,E2 28091.028} C_VEL
LIN {X 0,Y 601.037,Z 186.287,A -85,B 0,C 180,E1 28087.937,E2 28087.937} C_VEL
LIN {X 0,Y 601.107,Z 186.295,A -85,B 0,C 180,E1 28084.866,E2 28084.866} C_VEL
LIN {X 0,Y 601.039,Z 186.283,A -85,B 0,C 180,E1 28081.811,E2 28081.811} C_VEL
LIN {X 0,Y 601.075,Z 186.289,A -85,B 0,C 180,E1 28078.665,E2 28078.665} C_VEL
LIN {X 0,Y 601.049,Z 186.289,A -85,B 0,C 180,E1 28075.707,E2 28075.707} C_VEL
LIN {X 0,Y 601.048,Z 186.28,A -85,B 0,C 180,E1 28072.448,E2 28072.448} C_VEL
LIN {X 0,Y 601.067,Z 186.294,A -85,B 0,C 180,E1 28069.553,E2 28069.553} C_VEL
LIN {X 0,Y 601.045,Z 186.291,A -85,B 0,C 180,E1 28066.434,E2 28066.434} C_VEL
LIN {X 0,Y 601.063,Z 186.295,A -85,B 0,C 180,E1 28063.672,E2 28063.672} C_VEL
LIN {X 0,Y 601.044,Z 186.296,A -85,B 0,C 180,E1 28060.465,E2 28060.465} C_VEL
LIN {X 0,Y 601.087,Z 186.284,A -85,B 0,C 180,E1 28057.505,E2 28057.505} C_VEL
LIN {X 0,Y 601.041,Z 186.29,A -85,B 0,C 180,E1 28054.362,E2 28054.362} C_VEL
LIN {X 0,Y 601.112,Z 186.252,A -85,B 0,C 180,E1 28051.267,E2 28051.267} C_VEL
LIN {X 0,Y 601.042,Z 186.296,A -85,B 0,C 180,E1 28048.285,E2 28048.285} C_VEL
LIN {X 0,Y 601.092,Z 186.271,A -85,B 0,C 180,E1 28045.21,E2 28045.21} C_VEL
LIN {X 0,Y 601.043,Z 186.297,A -85,B 0,C 180,E1 28042.251,E2 28042.251} C_VEL
LIN {X 0,Y 601.083,Z 186.282,A -85,B 0,C 180,E1 28039.175,E2 28039.175} C_VEL
LIN {X 0,Y 601.048,Z 186.287,A -85,B 0,C 180,E1 28036.207,E2 28036.207} C_VEL
LIN {X 0,Y 601.049,Z 186.289,A -85,B 0,C 180,E1 28032.868,E2 28032.868} C_VEL
LIN {X 0,Y 601.062,Z 186.296,A -85,B 0,C 180,E1 28030.068,E2 28030.068} C_VEL
LIN {X 0,Y 601.04,Z 186.243,A -85,B 0,C 180,E1 28026.851,E2 28026.851} C_VEL
LIN {X 0,Y 601.103,Z 186.687,A -85,B 0,C 180,E1 28026.454,E2 28026.454} C_VEL
LIN {X 0,Y 607.72,Z 207.69,A -85,B 0,C 180,E1 28023.896,E2 28023.896} C_VEL
LIN {X 0,Y 611.329,Z 220.936,A -85,B 0,C 180,E1 28022.384,E2 28022.384} C_VEL
LIN {X 0,Y 611.208,Z 223.325,A -85,B 0,C 180,E1 28022.169,E2 28022.169} C_VEL
LIN {X 0,Y 618.292,Z 256.356,A -85,B 0,C 180,E1 28021.295,E2 28021.295} C_VEL
LIN {X 0,Y 614.617,Z 521.059,A -85,B 0,C 180,E1 28018.003,E2 28018.003} C_VEL
LIN {X 0,Y 614.041,Z 539.756,A -85,B 0,C 180,E1 28017.687,E2 28017.687} C_VEL
LIN {X 0,Y 613.325,Z 557.22,A -85,B 0,C 180,E1 28017.281,E2 28017.281} C_VEL
LIN {X 0,Y 612.494,Z 574.222,A -85,B 0,C 180,E1 28016.776,E2 28016.776} C_VEL
LIN {X 0,Y 611.566,Z 590.366,A -85,B 0,C 180,E1 28016.192,E2 28016.192} C_VEL
LIN {X 0,Y 610.489,Z 607.329,A -85,B 0,C 180,E1 28015.46,E2 28015.46} C_VEL
LIN {X 0,Y 609.096,Z 627.374,A -85,B 0,C 180,E1 28014.433,E2 28014.433} C_VEL
LIN {X 0,Y 607.64,Z 646.197,A -85,B 0,C 180,E1 28013.258,E2 28013.258} C_VEL
LIN {X 0,Y 606.453,Z 661.165,A -85,B 0,C 180,E1 28012.18,E2 28012.18} C_VEL
LIN {X 0,Y 605.341,Z 674.955,A -85,B 0,C 180,E1 28011.051,E2 28011.051} C_VEL
LIN {X 0,Y 604.348,Z 687.618,A -85,B 0,C 180,E1 28009.881,E2 28009.881} C_VEL
LIN {X 0,Y 603.401,Z 700.061,A -85,B 0,C 180,E1 28008.583,E2 28008.583} C_VEL
LIN {X 0,Y 602.534,Z 711.962,A -85,B 0,C 180,E1 28007.178,E2 28007.178} C_VEL
LIN {X 0,Y 601.688,Z 724.993,A -85,B 0,C 180,E1 28005.418,E2 28005.418} C_VEL
LIN {X 0,Y 601.01,Z 736.446,A -85,B 0,C 180,E1 28003.565,E2 28003.565} C_VEL
LIN {X 0,Y 600.583,Z 745.179,A -85,B 0,C 180,E1 28001.912,E2 28001.912} C_VEL
LIN {X 0,Y 600.31,Z 752.183,A -85,B 0,C 180,E1 28000.362,E2 28000.362} C_VEL
LIN {X 0,Y 600.111,Z 758.083,A -85,B 0,C 180,E1 27998.816,E2 27998.816} C_VEL
LIN {X 0,Y 600.002,Z 763.216,A -85,B 0,C 180,E1 27997.179,E2 27997.179} C_VEL
LIN {X 0,Y 599.945,Z 767.242,A -85,B 0,C 180,E1 27995.546,E2 27995.546} C_VEL
LIN {X 0,Y 599.924,Z 770.204,A -85,B 0,C 180,E1 27993.918,E2 27993.918} C_VEL
LIN {X 0,Y 599.912,Z 772.221,A -85,B 0,C 180,E1 27992.197,E2 27992.197} C_VEL
LIN {X 0,Y 599.907,Z 773.165,A -85,B 0,C 180,E1 27990.286,E2 27990.286} C_VEL
LIN {X 0,Y 599.916,Z 772.397,A -85,B 0,C 180,E1 27987.994,E2 27987.994} C_VEL
LIN {X 0,Y 599.923,Z 770.351,A -85,B 0,C 180,E1 27986.178,E2 27986.178} C_VEL
LIN {X 0,Y 599.942,Z 767.45,A -85,B 0,C 180,E1 27984.549,E2 27984.549} C_VEL
LIN {X 0,Y 599.993,Z 763.486,A -85,B 0,C 180,E1 27982.917,E2 27982.917} C_VEL
LIN {X 0,Y 600.102,Z 758.416,A -85,B 0,C 180,E1 27981.28,E2 27981.28} C_VEL
LIN {X 0,Y 600.295,Z 752.582,A -85,B 0,C 180,E1 27979.735,E2 27979.735} C_VEL
LIN {X 0,Y 600.562,Z 745.647,A -85,B 0,C 180,E1 27978.185,E2 27978.185} C_VEL
LIN {X 0,Y 600.944,Z 737.528,A -85,B 0,C 180,E1 27976.63,E2 27976.63} C_VEL
LIN {X 0,Y 601.526,Z 727.498,A -85,B 0,C 180,E1 27974.973,E2 27974.973} C_VEL
LIN {X 0,Y 602.477,Z 712.847,A -85,B 0,C 180,E1 27972.931,E2 27972.931} C_VEL
LIN {X 0,Y 603.378,Z 700.365,A -85,B 0,C 180,E1 27971.45,E2 27971.45} C_VEL
LIN {X 0,Y 604.306,Z 688.184,A -85,B 0,C 180,E1 27970.175,E2 27970.175} C_VEL
LIN {X 0,Y 605.299,Z 675.508,A -85,B 0,C 180,E1 27968.997,E2 27968.997} C_VEL
LIN {X 0,Y 606.401,Z 661.795,A -85,B 0,C 180,E1 27967.869,E2 27967.869} C_VEL
LIN {X 0,Y 607.58,Z 646.942,A -85,B 0,C 180,E1 27966.793,E2 27966.793} C_VEL
LIN {X 0,Y 609.029,Z 628.213,A -85,B 0,C 180,E1 27965.616,E2 27965.616} C_VEL
LIN {X 0,Y 610.422,Z 608.392,A -85,B 0,C 180,E1 27964.589,E2 27964.589} C_VEL
LIN {X 0,Y 611.494,Z 591.646,A -85,B 0,C 180,E1 27963.858,E2 27963.858} C_VEL
LIN {X 0,Y 612.44,Z 575.311,A -85,B 0,C 180,E1 27963.26,E2 27963.26} C_VEL
LIN {X 0,Y 613.292,Z 557.906,A -85,B 0,C 180,E1 27962.737,E2 27962.737} C_VEL
LIN {X 0,Y 614.009,Z 540.492,A -85,B 0,C 180,E1 27962.328,E2 27962.328} C_VEL
LIN {X 0,Y 614.573,Z 522.669,A -85,B 0,C 180,E1 27962.021,E2 27962.021} C_VEL
LIN {X 0,Y 618.195,Z 263.317,A -85,B 0,C 180,E1 27958.792,E2 27958.792} C_VEL
LIN {X 0,Y 618.114,Z 254.797,A -85,B 0,C 180,E1 27958.674,E2 27958.674} C_VEL
LIN {X 0,Y 611.206,Z 223.321,A -85,B 0,C 180,E1 27957.831,E2 27957.831} C_VEL
LIN {X 0,Y 611.212,Z 219.81,A -85,B 0,C 180,E1 27957.498,E2 27957.498} C_VEL
LIN {X 0,Y 605.241,Z 199.637,A -85,B 0,C 180,E1 27955.143,E2 27955.143} C_VEL
LIN {X 0,Y 601.059,Z 186.426,A -85,B 0,C 180,E1 27953.489,E2 27953.489} C_VEL
LIN {X 0,Y 601.087,Z 186.27,A -85,B 0,C 180,E1 27950.671,E2 27950.671} C_VEL
LIN {X 0,Y 601.041,Z 186.286,A -85,B 0,C 180,E1 27947.616,E2 27947.616} C_VEL
LIN {X 0,Y 601.106,Z 186.277,A -85,B 0,C 180,E1 27944.585,E2 27944.585} C_VEL
LIN {X 0,Y 601.04,Z 186.295,A -85,B 0,C 180,E1 27941.538,E2 27941.538} C_VEL
LIN {X 0,Y 601.11,Z 186.287,A -85,B 0,C 180,E1 27938.471,E2 27938.471} C_VEL
LIN {X 0,Y 601.041,Z 186.28,A -85,B 0,C 180,E1 27935.408,E2 27935.408} C_VEL
LIN {X 0,Y 601.078,Z 186.296,A -85,B 0,C 180,E1 27932.275,E2 27932.275} C_VEL
LIN {X 0,Y 601.043,Z 186.272,A -85,B 0,C 180,E1 27929.391,E2 27929.391} C_VEL
LIN {X 0,Y 601.058,Z 186.287,A -85,B 0,C 180,E1 27926.158,E2 27926.158} C_VEL
LIN {X 0,Y 601.063,Z 186.295,A -85,B 0,C 180,E1 27923.22,E2 27923.22} C_VEL
LIN {X 0,Y 601.043,Z 186.295,A -85,B 0,C 180,E1 27919.982,E2 27919.982} C_VEL
LIN {X 0,Y 601.097,Z 186.281,A -85,B 0,C 180,E1 27916.992,E2 27916.992} C_VEL
LIN {X 0,Y 601.04,Z 186.289,A -85,B 0,C 180,E1 27913.959,E2 27913.959} C_VEL
LIN {X 0,Y 601.108,Z 186.29,A -85,B 0,C 180,E1 27910.931,E2 27910.931} C_VEL
LIN {X 0,Y 601.038,Z 186.282,A -85,B 0,C 180,E1 27907.841,E2 27907.841} C_VEL
LIN {X 0,Y 601.098,Z 186.291,A -85,B 0,C 180,E1 27904.771,E2 27904.771} C_VEL
LIN {X 0,Y 601.043,Z 186.29,A -85,B 0,C 180,E1 27901.716,E2 27901.716} C_VEL
LIN {X 0,Y 601.056,Z 186.283,A -85,B 0,C 180,E1 27898.475,E2 27898.475} C_VEL
LIN {X 0,Y 601.053,Z 186.294,A -85,B 0,C 180,E1 27895.611,E2 27895.611} C_VEL
LIN {X 0,Y 601.044,Z 186.288,A -85,B 0,C 180,E1 27892.352,E2 27892.352} C_VEL
LIN {X 0,Y 601.083,Z 186.295,A -85,B 0,C 180,E1 27889.415,E2 27889.415} C_VEL
LIN {X 0,Y 601.039,Z 186.294,A -85,B 0,C 180,E1 27886.266,E2 27886.266} C_VEL
LIN {X 0,Y 601.106,Z 186.283,A -85,B 0,C 180,E1 27883.275,E2 27883.275} C_VEL
LIN {X 0,Y 601.038,Z 186.295,A -85,B 0,C 180,E1 27880.262,E2 27880.262} C_VEL
LIN {X 0,Y 601.116,Z 186.289,A -85,B 0,C 180,E1 27877.197,E2 27877.197} C_VEL
LIN {X 0,Y 601.04,Z 186.285,A -85,B 0,C 180,E1 27874.143,E2 27874.143} C_VEL
LIN {X 0,Y 601.069,Z 186.268,A -85,B 0,C 180,E1 27870.938,E2 27870.938} C_VEL
LIN {X 0,Y 601.046,Z 186.297,A -85,B 0,C 180,E1 27868.061,E2 27868.061} C_VEL
LIN {X 0,Y 601.043,Z 186.264,A -85,B 0,C 180,E1 27864.741,E2 27864.741} C_VEL
LIN {X 0,Y 601.075,Z 186.295,A -85,B 0,C 180,E1 27861.77,E2 27861.77} C_VEL
LIN {X 0,Y 601.045,Z 186.296,A -85,B 0,C 180,E1 27858.666,E2 27858.666} C_VEL
LIN {X 0,Y 601.099,Z 186.296,A -85,B 0,C 180,E1 27855.658,E2 27855.658} C_VEL
LIN {X 0,Y 601.039,Z 186.297,A -85,B 0,C 180,E1 27852.525,E2 27852.525} C_VEL
LIN {X 0,Y 601.108,Z 186.293,A -85,B 0,C 180,E1 27849.445,E2 27849.445} C_VEL
LIN {X 0,Y 601.041,Z 186.297,A -85,B 0,C 180,E1 27846.429,E2 27846.429} C_VEL
LIN {X 0,Y 601.079,Z 186.298,A -85,B 0,C 180,E1 27843.29,E2 27843.29} C_VEL
LIN {X 0,Y 601.045,Z 186.297,A -85,B 0,C 180,E1 27840.375,E2 27840.375} C_VEL
LIN {X 0,Y 601.056,Z 186.299,A -85,B 0,C 180,E1 27838.233,E2 27838.233} C_VEL
LIN {X 0,Y 600.112,Z 186.419,A -85,B 0,C 180,E1 27837.498,E2 27837.498} C_VEL
LIN {X 0,Y 593.562,Z 187.233,A -85,B 0,C 180,E1 27835.385,E2 27835.385} C_VEL
LIN {X 0,Y 593.105,Z 187.288,A -85,B 0,C 180,E1 27834.901,E2 27834.901} C_VEL
LIN {X 0,Y 593.181,Z 187.283,A -85,B 0,C 180,E1 27831.753,E2 27831.753} C_VEL
LIN {X 0,Y 593.102,Z 187.289,A -85,B 0,C 180,E1 27828.655,E2 27828.655} C_VEL
LIN {X 0,Y 593.143,Z 187.284,A -85,B 0,C 180,E1 27825.545,E2 27825.545} C_VEL
LIN {X 0,Y 593.101,Z 187.287,A -85,B 0,C 180,E1 27822.658,E2 27822.658} C_VEL
LIN {X 0,Y 593.122,Z 187.288,A -85,B 0,C 180,E1 27819.41,E2 27819.41} C_VEL
LIN {X 0,Y 593.108,Z 187.29,A -85,B 0,C 180,E1 27816.582,E2 27816.582} C_VEL
LIN {X 0,Y 593.107,Z 187.288,A -85,B 0,C 180,E1 27813.285,E2 27813.285} C_VEL
LIN {X 0,Y 593.141,Z 187.285,A -85,B 0,C 180,E1 27810.29,E2 27810.29} C_VEL
LIN {X 0,Y 593.101,Z 187.29,A -85,B 0,C 180,E1 27807.198,E2 27807.198} C_VEL
LIN {X 0,Y 593.174,Z 187.281,A -85,B 0,C 180,E1 27804.099,E2 27804.099} C_VEL
LIN {X 0,Y 593.099,Z 187.287,A -85,B 0,C 180,E1 27801.079,E2 27801.079} C_VEL
LIN {X 0,Y 593.155,Z 187.286,A -85,B 0,C 180,E1 27797.936,E2 27797.936} C_VEL
LIN {X 0,Y 593.104,Z 187.29,A -85,B 0,C 180,E1 27794.954,E2 27794.954} C_VEL
LIN {X 0,Y 593.125,Z 187.286,A -85,B 0,C 180,E1 27791.729,E2 27791.729} C_VEL
LIN {X 0,Y 593.117,Z 187.286,A -85,B 0,C 180,E1 27788.79,E2 27788.79} C_VEL
LIN {X 0,Y 593.106,Z 187.289,A -85,B 0,C 180,E1 27785.502,E2 27785.502} C_VEL
LIN {X 0,Y 593.17,Z 187.283,A -85,B 0,C 180,E1 27782.387,E2 27782.387} C_VEL
LIN {X 0,Y 593.099,Z 187.287,A -85,B 0,C 180,E1 27779.286,E2 27779.286} C_VEL
LIN {X 0,Y 593.157,Z 187.284,A -85,B 0,C 180,E1 27776.206,E2 27776.206} C_VEL
LIN {X 0,Y 593.108,Z 187.286,A -85,B 0,C 180,E1 27773.124,E2 27773.124} C_VEL
LIN {X 0,Y 593.112,Z 187.286,A -85,B 0,C 180,E1 27769.79,E2 27769.79} C_VEL
LIN {X 0,Y 593.131,Z 187.286,A -85,B 0,C 180,E1 27766.882,E2 27766.882} C_VEL
LIN {X 0,Y 593.103,Z 187.286,A -85,B 0,C 180,E1 27763.686,E2 27763.686} C_VEL
LIN {X 0,Y 593.178,Z 187.283,A -85,B 0,C 180,E1 27760.592,E2 27760.592} C_VEL
LIN {X 0,Y 593.099,Z 187.284,A -85,B 0,C 180,E1 27757.604,E2 27757.604} C_VEL
LIN {X 0,Y 593.158,Z 187.249,A -85,B 0,C 180,E1 27754.493,E2 27754.493} C_VEL
LIN {X 0,Y 593.104,Z 187.286,A -85,B 0,C 180,E1 27751.468,E2 27751.468} C_VEL
LIN {X 0,Y 593.137,Z 187.237,A -85,B 0,C 180,E1 27748.376,E2 27748.376} C_VEL
LIN {X 0,Y 593.113,Z 187.273,A -85,B 0,C 180,E1 27745.354,E2 27745.354} C_VEL
LIN {X 0,Y 593.108,Z 187.275,A -85,B 0,C 180,E1 27742.083,E2 27742.083} C_VEL
LIN {X 0,Y 593.145,Z 187.284,A -85,B 0,C 180,E1 27739.089,E2 27739.089} C_VEL
LIN {X 0,Y 593.1,Z 187.28,A -85,B 0,C 180,E1 27735.95,E2 27735.95} C_VEL
LIN {X 0,Y 593.167,Z 187.271,A -85,B 0,C 180,E1 27732.956,E2 27732.956} C_VEL
LIN {X 0,Y 593.101,Z 187.284,A -85,B 0,C 180,E1 27729.804,E2 27729.804} C_VEL
LIN {X 0,Y 593.148,Z 187.275,A -85,B 0,C 180,E1 27726.68,E2 27726.68} C_VEL
LIN {X 0,Y 593.106,Z 187.284,A -85,B 0,C 180,E1 27723.673,E2 27723.673} C_VEL
LIN {X 0,Y 593.112,Z 187.284,A -85,B 0,C 180,E1 27720.386,E2 27720.386} C_VEL
LIN {X 0,Y 593.125,Z 187.276,A -85,B 0,C 180,E1 27717.488,E2 27717.488} C_VEL
LIN {X 0,Y 593.104,Z 187.282,A -85,B 0,C 180,E1 27714.292,E2 27714.292} C_VEL
LIN {X 0,Y 593.158,Z 187.268,A -85,B 0,C 180,E1 27711.274,E2 27711.274} C_VEL
LIN {X 0,Y 593.1,Z 187.278,A -85,B 0,C 180,E1 27708.131,E2 27708.131} C_VEL
LIN {X 0,Y 593.168,Z 187.284,A -85,B 0,C 180,E1 27705.054,E2 27705.054} C_VEL
LIN {X 0,Y 593.103,Z 187.273,A -85,B 0,C 180,E1 27702.03,E2 27702.03} C_VEL
LIN {X 0,Y 593.132,Z 187.275,A -85,B 0,C 180,E1 27698.853,E2 27698.853} C_VEL
LIN {X 0,Y 593.109,Z 187.284,A -85,B 0,C 180,E1 27696.008,E2 27696.008} C_VEL
LIN {X 0,Y 593.111,Z 187.251,A -85,B 0,C 180,E1 27692.706,E2 27692.706} C_VEL
LIN {X 0,Y 593.121,Z 187.267,A -85,B 0,C 180,E1 27689.843,E2 27689.843} C_VEL
LIN {X 0,Y 593.107,Z 187.277,A -85,B 0,C 180,E1 27686.661,E2 27686.661} C_VEL
LIN {X 0,Y 593.157,Z 187.271,A -85,B 0,C 180,E1 27683.603,E2 27683.603} C_VEL
LIN {X 0,Y 593.1,Z 187.271,A -85,B 0,C 180,E1 27680.536,E2 27680.536} C_VEL
LIN {X 0,Y 593.174,Z 187.281,A -85,B 0,C 180,E1 27677.472,E2 27677.472} C_VEL
LIN {X 0,Y 593.103,Z 187.285,A -85,B 0,C 180,E1 27674.372,E2 27674.372} C_VEL
LIN {X 0,Y 593.142,Z 187.278,A -85,B 0,C 180,E1 27671.227,E2 27671.227} C_VEL
LIN {X 0,Y 593.1,Z 187.232,A -85,B 0,C 180,E1 27668.339,E2 27668.339} C_VEL
LIN {X 0,Y 593.146,Z 187.524,A -85,B 0,C 180,E1 27666.916,E2 27666.916} C_VEL
LIN {X 0,Y 598.981,Z 205.857,A -85,B 0,C 180,E1 27664.616,E2 27664.616} C_VEL
LIN {X 0,Y 603.928,Z 222.898,A -85,B 0,C 180,E1 27662.615,E2 27662.615} C_VEL
LIN {X 0,Y 606.947,Z 236.538,A -85,B 0,C 180,E1 27662.215,E2 27662.215} C_VEL
LIN {X 0,Y 611.423,Z 258.062,A -85,B 0,C 180,E1 27661.662,E2 27661.662} C_VEL
